LIN {X 0,Y 235.398,Z 339.465,A -85,B 0,C 180,E1 -19978.483,E2 -19978.483} C_VEL
LIN {X 0,Y 236.416,Z 340.763,A -85,B 0,C 180,E1 -19979.023,E2 -19979.023} C_VEL
LIN {X 0,Y 240.93,Z 348.91,A -85,B 0,C 180,E1 -19981.671,E2 -19981.671} C_VEL
LIN {X 0,Y 245.217,Z 358.248,A -85,B 0,C 180,E1 -19984.418,E2 -19984.418} C_VEL
LIN {X 0,Y 247.633,Z 366.708,A -85,B 0,C 180,E1 -19986.619,E2 -19986.619} C_VEL
LIN {X 0,Y 248.994,Z 374.297,A -85,B 0,C 180,E1 -19988.522,E2 -19988.522} C_VEL
LIN {X 0,Y 249.236,Z 377.337,A -85,B 0,C 180,E1 -19989.268,E2 -19989.268} C_VEL
LIN {X 0,Y 246.011,Z 387.134,A -85,B 0,C 180,E1 -19991.118,E2 -19991.118} C_VEL
LIN {X 0,Y 242.427,Z 396.773,A -85,B 0,C 180,E1 -19993.41,E2 -19993.41} C_VEL
LIN {X 0,Y 239.164,Z 404.642,A -85,B 0,C 180,E1 -19995.772,E2 -19995.772} C_VEL
LIN {X 0,Y 236.021,Z 411.635,A -85,B 0,C 180,E1 -19998.498,E2 -19998.498} C_VEL
LIN {X 0,Y 233.343,Z 416.972,A -85,B 0,C 180,E1 -20001.188,E2 -20001.188} C_VEL
LIN {X 0,Y 231.011,Z 421.302,A -85,B 0,C 180,E1 -20004.12,E2 -20004.12} C_VEL
LIN {X 0,Y 229.008,Z 424.571,A -85,B 0,C 180,E1 -20007.408,E2 -20007.408} C_VEL
LIN {X 0,Y 227.709,Z 426.199,A -85,B 0,C 180,E1 -20010.209,E2 -20010.209} C_VEL
LIN {X 0,Y 226.788,Z 426.825,A -85,B 0,C 180,E1 -20013.205,E2 -20013.205} C_VEL
LIN {X 0,Y 226.233,Z 426.352,A -85,B 0,C 180,E1 -20016.174,E2 -20016.174} C_VEL
LIN {X 0,Y 226.037,Z 424.901,A -85,B 0,C 180,E1 -20018.985,E2 -20018.985} C_VEL
LIN {X 0,Y 226.222,Z 422.441,A -85,B 0,C 180,E1 -20021.788,E2 -20021.788} C_VEL
LIN {X 0,Y 226.652,Z 419.03,A -85,B 0,C 180,E1 -20024.505,E2 -20024.505} C_VEL
LIN {X 0,Y 227.314,Z 414.656,A -85,B 0,C 180,E1 -20027.141,E2 -20027.141} C_VEL
LIN {X 0,Y 228.15,Z 409.299,A -85,B 0,C 180,E1 -20029.692,E2 -20029.692} C_VEL
LIN {X 0,Y 229.267,Z 402.802,A -85,B 0,C 180,E1 -20032.187,E2 -20032.187} C_VEL
LIN {X 0,Y 230.625,Z 395.016,A -85,B 0,C 180,E1 -20034.619,E2 -20034.619} C_VEL
LIN {X 0,Y 232.373,Z 385.49,A -85,B 0,C 180,E1 -20037.016,E2 -20037.016} C_VEL
LIN {X 0,Y 234.011,Z 375.473,A -85,B 0,C 180,E1 -20039.048,E2 -20039.048} C_VEL
LIN {X 0,Y 235.622,Z 365.003,A -85,B 0,C 180,E1 -20040.768,E2 -20040.768} C_VEL
LIN {X 0,Y 236.33,Z 359.176,A -85,B 0,C 180,E1 -20041.588,E2 -20041.588} C_VEL
LIN {X 0,Y 234.059,Z 347.494,A -85,B 0,C 180,E1 -20043.23,E2 -20043.23} C_VEL
LIN {X 0,Y 230.539,Z 335.099,A -85,B 0,C 180,E1 -20044.736,E2 -20044.736} C_VEL
LIN {X 0,Y 227.695,Z 326.123,A -85,B 0,C 180,E1 -20045.678,E2 -20045.678} C_VEL
LIN {X 0,Y 227.868,Z 326.101,A -85,B 0,C 180,E1 -20048.277,E2 -20048.277} C_VEL
LIN {X 0,Y 227.99,Z 326.086,A -85,B 0,C 180,E1 -20052.862,E2 -20052.862} C_VEL
LIN {X 0,Y 228.066,Z 326.077,A -85,B 0,C 180,E1 -20057.543,E2 -20057.543} C_VEL
LIN {X 0,Y 228.259,Z 326.056,A -85,B 0,C 180,E1 -20061.144,E2 -20061.144} C_VEL
LIN {X 0,Y 228.31,Z 326.047,A -85,B 0,C 180,E1 -20062.927,E2 -20062.927} C_VEL
LIN {X 0,Y 228.554,Z 326.015,A -85,B 0,C 180,E1 -20068.238,E2 -20068.238} C_VEL
LIN {X 0,Y 228.555,Z 326.011,A -85,B 0,C 180,E1 -20071.762,E2 -20071.762} C_VEL
LIN {X 0,Y 228.31,Z 326.043,A -85,B 0,C 180,E1 -20077.073,E2 -20077.073} C_VEL
LIN {X 0,Y 228.146,Z 326.068,A -85,B 0,C 180,E1 -20080.651,E2 -20080.651} C_VEL
LIN {X 0,Y 228.066,Z 326.076,A -85,B 0,C 180,E1 -20084.272,E2 -20084.272} C_VEL
LIN {X 0,Y 228.004,Z 326.083,A -85,B 0,C 180,E1 -20087.953,E2 -20087.953} C_VEL
LIN {X 0,Y 227.931,Z 326.092,A -85,B 0,C 180,E1 -20092.33,E2 -20092.33} C_VEL
LIN {X 0,Y 227.944,Z 326.091,A -85,B 0,C 180,E1 -20096.603,E2 -20096.603} C_VEL
LIN {X 0,Y 227.91,Z 326.094,A -85,B 0,C 180,E1 -20100.296,E2 -20100.296} C_VEL
LIN {X 0,Y 227.889,Z 326.098,A -85,B 0,C 180,E1 -20103.719,E2 -20103.719} C_VEL
LIN {X 0,Y 227.87,Z 326.099,A -85,B 0,C 180,E1 -20108.086,E2 -20108.086} C_VEL
LIN {X 0,Y 227.815,Z 326.106,A -85,B 0,C 180,E1 -20112.742,E2 -20112.742} C_VEL
LIN {X 0,Y 227.812,Z 326.104,A -85,B 0,C 180,E1 -20117.258,E2 -20117.258} C_VEL
LIN {X 0,Y 227.846,Z 326.103,A -85,B 0,C 180,E1 -20121.91,E2 -20121.91} C_VEL
LIN {X 0,Y 227.887,Z 326.095,A -85,B 0,C 180,E1 -20126.375,E2 -20126.375} C_VEL
LIN {X 0,Y 227.921,Z 326.092,A -85,B 0,C 180,E1 -20130.438,E2 -20130.438} C_VEL
LIN {X 0,Y 227.927,Z 326.09,A -85,B 0,C 180,E1 -20134.426,E2 -20134.426} C_VEL
LIN {X 0,Y 227.947,Z 326.089,A -85,B 0,C 180,E1 -20138.286,E2 -20138.286} C_VEL
LIN {X 0,Y 228.011,Z 326.081,A -85,B 0,C 180,E1 -20142.848,E2 -20142.848} C_VEL
LIN {X 0,Y 228.06,Z 326.075,A -85,B 0,C 180,E1 -20147.543,E2 -20147.543} C_VEL
LIN {X 0,Y 228.267,Z 326.052,A -85,B 0,C 180,E1 -20151.145,E2 -20151.145} C_VEL
LIN {X 0,Y 228.322,Z 326.045,A -85,B 0,C 180,E1 -20152.928,E2 -20152.928} C_VEL
LIN {X 0,Y 228.556,Z 326.011,A -85,B 0,C 180,E1 -20158.238,E2 -20158.238} C_VEL
LIN {X 0,Y 228.552,Z 326.014,A -85,B 0,C 180,E1 -20161.762,E2 -20161.762} C_VEL
LIN {X 0,Y 228.312,Z 326.044,A -85,B 0,C 180,E1 -20167.073,E2 -20167.073} C_VEL
LIN {X 0,Y 228.148,Z 326.068,A -85,B 0,C 180,E1 -20170.651,E2 -20170.651} C_VEL
LIN {X 0,Y 228.051,Z 326.075,A -85,B 0,C 180,E1 -20174.273,E2 -20174.273} C_VEL
LIN {X 0,Y 227.972,Z 326.087,A -85,B 0,C 180,E1 -20177.956,E2 -20177.956} C_VEL
LIN {X 0,Y 227.923,Z 326.091,A -85,B 0,C 180,E1 -20182.323,E2 -20182.323} C_VEL
LIN {X 0,Y 227.926,Z 326.081,A -85,B 0,C 180,E1 -20186.593,E2 -20186.593} C_VEL
LIN {X 0,Y 227.877,Z 326.097,A -85,B 0,C 180,E1 -20190.281,E2 -20190.281} C_VEL
LIN {X 0,Y 227.89,Z 326.098,A -85,B 0,C 180,E1 -20193.719,E2 -20193.719} C_VEL
LIN {X 0,Y 227.871,Z 326.102,A -85,B 0,C 180,E1 -20198.086,E2 -20198.086} C_VEL
LIN {X 0,Y 227.925,Z 326.208,A -85,B 0,C 180,E1 -20199.568,E2 -20199.568} C_VEL
LIN {X 0,Y 228.797,Z 330.781,A -85,B 0,C 180,E1 -20203.721,E2 -20203.721} C_VEL
LIN {X 0,Y 229.869,Z 336.683,A -85,B 0,C 180,E1 -20208.812,E2 -20208.812} C_VEL
LIN {X 0,Y 230.393,Z 339.72,A -85,B 0,C 180,E1 -20211.293,E2 -20211.293} C_VEL
LIN {X 0,Y 230.3,Z 342.542,A -85,B 0,C 180,E1 -20213.506,E2 -20213.506} C_VEL
LIN {X 0,Y 228.77,Z 349.178,A -85,B 0,C 180,E1 -20218.516,E2 -20218.516} C_VEL
LIN {X 0,Y 228.509,Z 350.58,A -85,B 0,C 180,E1 -20219.558,E2 -20219.558} C_VEL
LIN {X 0,Y 228.015,Z 352.382,A -85,B 0,C 180,E1 -20220.39,E2 -20220.39} C_VEL
LIN {X 0,Y 227.044,Z 355.768,A -85,B 0,C 180,E1 -20221.22,E2 -20221.22} C_VEL
LIN {X 0,Y 225.918,Z 359.881,A -85,B 0,C 180,E1 -20221.849,E2 -20221.849} C_VEL
LIN {X 0,Y 224.603,Z 365.585,A -85,B 0,C 180,E1 -20222.423,E2 -20222.423} C_VEL
LIN {X 0,Y 223.56,Z 373.659,A -85,B 0,C 180,E1 -20223.095,E2 -20223.095} C_VEL
LIN {X 0,Y 223.654,Z 377.387,A -85,B 0,C 180,E1 -20223.476,E2 -20223.476} C_VEL
LIN {X 0,Y 224.58,Z 389.329,A -85,B 0,C 180,E1 -20224.966,E2 -20224.966} C_VEL
LIN {X 0,Y 225.134,Z 401.195,A -85,B 0,C 180,E1 -20226.789,E2 -20226.789} C_VEL
LIN {X 0,Y 225.215,Z 410.46,A -85,B 0,C 180,E1 -20228.49,E2 -20228.49} C_VEL
LIN {X 0,Y 223.359,Z 420.599,A -85,B 0,C 180,E1 -20230.662,E2 -20230.662} C_VEL
LIN {X 0,Y 221.808,Z 429.212,A -85,B 0,C 180,E1 -20232.957,E2 -20232.957} C_VEL
LIN {X 0,Y 220.521,Z 437.46,A -85,B 0,C 180,E1 -20235.7,E2 -20235.7} C_VEL
LIN {X 0,Y 219.699,Z 443.077,A -85,B 0,C 180,E1 -20237.999,E2 -20237.999} C_VEL
LIN {X 0,Y 219.222,Z 448.554,A -85,B 0,C 180,E1 -20240.776,E2 -20240.776} C_VEL
LIN {X 0,Y 219.119,Z 453.231,A -85,B 0,C 180,E1 -20243.878,E2 -20243.878} C_VEL
LIN {X 0,Y 219.084,Z 455.908,A -85,B 0,C 180,E1 -20246.321,E2 -20246.321} C_VEL
LIN {X 0,Y 219.205,Z 457.414,A -85,B 0,C 180,E1 -20248.163,E2 -20248.163} C_VEL
LIN {X 0,Y 219.481,Z 458.495,A -85,B 0,C 180,E1 -20250,E2 -20250} C_VEL
LIN {X 0,Y 218.947,Z 459.218,A -85,B 0,C 180,E1 -20253.681,E2 -20253.681} C_VEL
LIN {X 0,Y 218.814,Z 458.388,A -85,B 0,C 180,E1 -20257.382,E2 -20257.382} C_VEL
LIN {X 0,Y 219.34,Z 455.952,A -85,B 0,C 180,E1 -20261.084,E2 -20261.084} C_VEL
LIN {X 0,Y 220.319,Z 453.09,A -85,B 0,C 180,E1 -20263.842,E2 -20263.842} C_VEL
LIN {X 0,Y 222.516,Z 447.791,A -85,B 0,C 180,E1 -20267.461,E2 -20267.461} C_VEL
LIN {X 0,Y 225.054,Z 441.83,A -85,B 0,C 180,E1 -20270.471,E2 -20270.471} C_VEL
LIN {X 0,Y 227.921,Z 434.999,A -85,B 0,C 180,E1 -20273.151,E2 -20273.151} C_VEL
LIN {X 0,Y 231.455,Z 426.902,A -85,B 0,C 180,E1 -20275.639,E2 -20275.639} C_VEL
LIN {X 0,Y 233.903,Z 420.63,A -85,B 0,C 180,E1 -20277.272,E2 -20277.272} C_VEL
LIN {X 0,Y 236.072,Z 410.799,A -85,B 0,C 180,E1 -20279.626,E2 -20279.626} C_VEL
LIN {X 0,Y 237.181,Z 401.09,A -85,B 0,C 180,E1 -20281.733,E2 -20281.733} C_VEL
LIN {X 0,Y 237.255,Z 388.964,A -85,B 0,C 180,E1 -20284.251,E2 -20284.251} C_VEL
LIN {X 0,Y 236.12,Z 377.783,A -85,B 0,C 180,E1 -20286.534,E2 -20286.534} C_VEL
LIN {X 0,Y 233.941,Z 366.022,A -85,B 0,C 180,E1 -20289.016,E2 -20289.016} C_VEL
LIN {X 0,Y 232.372,Z 361.024,A -85,B 0,C 180,E1 -20290.209,E2 -20290.209} C_VEL
LIN {X 0,Y 230.909,Z 357.222,A -85,B 0,C 180,E1 -20291.235,E2 -20291.235} C_VEL
LIN {X 0,Y 228.734,Z 353.288,A -85,B 0,C 180,E1 -20292.567,E2 -20292.567} C_VEL
LIN {X 0,Y 227.831,Z 351.073,A -85,B 0,C 180,E1 -20293.186,E2 -20293.186} C_VEL
LIN {X 0,Y 225.159,Z 347.328,A -85,B 0,C 180,E1 -20294.836,E2 -20294.836} C_VEL
LIN {X 0,Y 224.055,Z 344.226,A -85,B 0,C 180,E1 -20295.74,E2 -20295.74} C_VEL
LIN {X 0,Y 223.573,Z 341.782,A -85,B 0,C 180,E1 -20298.977,E2 -20298.977} C_VEL
LIN {X 0,Y 223.1,Z 338.961,A -85,B 0,C 180,E1 -20303.235,E2 -20303.235} C_VEL
LIN {X 0,Y 222.676,Z 336.61,A -85,B 0,C 180,E1 -20307.551,E2 -20307.551} C_VEL
LIN {X 0,Y 222.34,Z 334.59,A -85,B 0,C 180,E1 -20312.26,E2 -20312.26} C_VEL
LIN {X 0,Y 222.116,Z 333.25,A -85,B 0,C 180,E1 -20316.578,E2 -20316.578} C_VEL
LIN {X 0,Y 221.976,Z 332.239,A -85,B 0,C 180,E1 -20321.776,E2 -20321.776} C_VEL
LIN {X 0,Y 221.961,Z 331.908,A -85,B 0,C 180,E1 -20325.326,E2 -20325.326} C_VEL
LIN {X 0,Y 222.119,Z 331.932,A -85,B 0,C 180,E1 -20330.897,E2 -20330.897} C_VEL
LIN {X 0,Y 222.172,Z 332.099,A -85,B 0,C 180,E1 -20331.472,E2 -20331.472} C_VEL
LIN {X 0,Y 223.328,Z 334.532,A -85,B 0,C 180,E1 -20332.484,E2 -20332.484} C_VEL
LIN {X 0,Y 225.884,Z 336.883,A -85,B 0,C 180,E1 -20334.131,E2 -20334.131} C_VEL
LIN {X 0,Y 228.082,Z 340.42,A -85,B 0,C 180,E1 -20335.692,E2 -20335.692} C_VEL
LIN {X 0,Y 229.492,Z 341.637,A -85,B 0,C 180,E1 -20336.488,E2 -20336.488} C_VEL
LIN {X 0,Y 232.052,Z 345.542,A -85,B 0,C 180,E1 -20338.113,E2 -20338.113} C_VEL
LIN {X 0,Y 235.66,Z 352.189,A -85,B 0,C 180,E1 -20340.512,E2 -20340.512} C_VEL
LIN {X 0,Y 239.595,Z 360.989,A -85,B 0,C 180,E1 -20343.363,E2 -20343.363} C_VEL
LIN {X 0,Y 241.713,Z 368.228,A -85,B 0,C 180,E1 -20345.422,E2 -20345.422} C_VEL
LIN {X 0,Y 243.137,Z 376.852,A -85,B 0,C 180,E1 -20347.765,E2 -20347.765} C_VEL
LIN {X 0,Y 243.302,Z 379.462,A -85,B 0,C 180,E1 -20348.448,E2 -20348.448} C_VEL
LIN {X 0,Y 239.625,Z 389.997,A -85,B 0,C 180,E1 -20350.562,E2 -20350.562} C_VEL
LIN {X 0,Y 235.887,Z 399.194,A -85,B 0,C 180,E1 -20352.911,E2 -20352.911} C_VEL
LIN {X 0,Y 232.47,Z 406.649,A -85,B 0,C 180,E1 -20355.328,E2 -20355.328} C_VEL
LIN {X 0,Y 229.237,Z 413.358,A -85,B 0,C 180,E1 -20358.119,E2 -20358.119} C_VEL
LIN {X 0,Y 226.177,Z 418.961,A -85,B 0,C 180,E1 -20361.22,E2 -20361.22} C_VEL
LIN {X 0,Y 223.73,Z 423.003,A -85,B 0,C 180,E1 -20364.359,E2 -20364.359} C_VEL
LIN {X 0,Y 221.864,Z 425.675,A -85,B 0,C 180,E1 -20367.506,E2 -20367.506} C_VEL
LIN {X 0,Y 220.445,Z 427.13,A -85,B 0,C 180,E1 -20370.67,E2 -20370.67} C_VEL
LIN {X 0,Y 219.586,Z 427.399,A -85,B 0,C 180,E1 -20373.679,E2 -20373.679} C_VEL
LIN {X 0,Y 219.082,Z 426.619,A -85,B 0,C 180,E1 -20376.68,E2 -20376.68} C_VEL
LIN {X 0,Y 218.979,Z 424.565,A -85,B 0,C 180,E1 -20379.933,E2 -20379.933} C_VEL
LIN {X 0,Y 219.391,Z 420.77,A -85,B 0,C 180,E1 -20383.551,E2 -20383.551} C_VEL
LIN {X 0,Y 219.954,Z 416.899,A -85,B 0,C 180,E1 -20386.181,E2 -20386.181} C_VEL
LIN {X 0,Y 220.89,Z 411.056,A -85,B 0,C 180,E1 -20389.257,E2 -20389.257} C_VEL
LIN {X 0,Y 222.145,Z 403.613,A -85,B 0,C 180,E1 -20392.272,E2 -20392.272} C_VEL
LIN {X 0,Y 223.574,Z 395.754,A -85,B 0,C 180,E1 -20394.816,E2 -20394.816} C_VEL
LIN {X 0,Y 225.395,Z 386.048,A -85,B 0,C 180,E1 -20397.339,E2 -20397.339} C_VEL
LIN {X 0,Y 227.175,Z 375.569,A -85,B 0,C 180,E1 -20399.517,E2 -20399.517} C_VEL
LIN {X 0,Y 228.882,Z 364.732,A -85,B 0,C 180,E1 -20401.329,E2 -20401.329} C_VEL
LIN {X 0,Y 229.386,Z 360.768,A -85,B 0,C 180,E1 -20401.896,E2 -20401.896} C_VEL
LIN {X 0,Y 227.646,Z 350.635,A -85,B 0,C 180,E1 -20403.407,E2 -20403.407} C_VEL
LIN {X 0,Y 224.857,Z 340.173,A -85,B 0,C 180,E1 -20404.795,E2 -20404.795} C_VEL
LIN {X 0,Y 220.665,Z 326.998,A -85,B 0,C 180,E1 -20406.291,E2 -20406.291} C_VEL
LIN {X 0,Y 220.829,Z 326.979,A -85,B 0,C 180,E1 -20409.508,E2 -20409.508} C_VEL
LIN {X 0,Y 220.978,Z 326.96,A -85,B 0,C 180,E1 -20413.367,E2 -20413.367} C_VEL
LIN {X 0,Y 221.003,Z 326.959,A -85,B 0,C 180,E1 -20417.138,E2 -20417.138} C_VEL
LIN {X 0,Y 221.199,Z 326.936,A -85,B 0,C 180,E1 -20420.859,E2 -20420.859} C_VEL
LIN {X 0,Y 221.13,Z 326.939,A -85,B 0,C 180,E1 -20424.529,E2 -20424.529} C_VEL
LIN {X 0,Y 221.512,Z 326.892,A -85,B 0,C 180,E1 -20428.182,E2 -20428.182} C_VEL
LIN {X 0,Y 221.512,Z 326.888,A -85,B 0,C 180,E1 -20431.818,E2 -20431.818} C_VEL
LIN {X 0,Y 221.247,Z 326.922,A -85,B 0,C 180,E1 -20437.3,E2 -20437.3} C_VEL
LIN {X 0,Y 221.068,Z 326.947,A -85,B 0,C 180,E1 -20440.996,E2 -20440.996} C_VEL
LIN {X 0,Y 220.997,Z 326.955,A -85,B 0,C 180,E1 -20444.739,E2 -20444.739} C_VEL
LIN {X 0,Y 220.923,Z 326.966,A -85,B 0,C 180,E1 -20448.549,E2 -20448.549} C_VEL
LIN {X 0,Y 220.897,Z 326.967,A -85,B 0,C 180,E1 -20452.683,E2 -20452.683} C_VEL
LIN {X 0,Y 220.887,Z 326.969,A -85,B 0,C 180,E1 -20457.016,E2 -20457.016} C_VEL
LIN {X 0,Y 220.864,Z 326.969,A -85,B 0,C 180,E1 -20460.779,E2 -20460.779} C_VEL
LIN {X 0,Y 220.815,Z 326.977,A -85,B 0,C 180,E1 -20464.953,E2 -20464.953} C_VEL
LIN {X 0,Y 220.839,Z 326.974,A -85,B 0,C 180,E1 -20467.288,E2 -20467.288} C_VEL
LIN {X 0,Y 220.776,Z 326.986,A -85,B 0,C 180,E1 -20471.952,E2 -20471.952} C_VEL
LIN {X 0,Y 220.775,Z 326.984,A -85,B 0,C 180,E1 -20475.546,E2 -20475.546} C_VEL
LIN {X 0,Y 220.808,Z 326.979,A -85,B 0,C 180,E1 -20480.464,E2 -20480.464} C_VEL
LIN {X 0,Y 220.807,Z 326.976,A -85,B 0,C 180,E1 -20485.046,E2 -20485.046} C_VEL
LIN {X 0,Y 220.87,Z 326.974,A -85,B 0,C 180,E1 -20489.395,E2 -20489.395} C_VEL
LIN {X 0,Y 220.897,Z 326.968,A -85,B 0,C 180,E1 -20493.55,E2 -20493.55} C_VEL
LIN {X 0,Y 220.867,Z 326.973,A -85,B 0,C 180,E1 -20497.552,E2 -20497.552} C_VEL
LIN {X 0,Y 220.965,Z 326.957,A -85,B 0,C 180,E1 -20502.59,E2 -20502.59} C_VEL
LIN {X 0,Y 220.999,Z 326.957,A -85,B 0,C 180,E1 -20507.138,E2 -20507.138} C_VEL
LIN {X 0,Y 221.205,Z 326.929,A -85,B 0,C 180,E1 -20510.86,E2 -20510.86} C_VEL
LIN {X 0,Y 221.258,Z 326.924,A -85,B 0,C 180,E1 -20512.701,E2 -20512.701} C_VEL
LIN {X 0,Y 221.514,Z 326.888,A -85,B 0,C 180,E1 -20518.182,E2 -20518.182} C_VEL
LIN {X 0,Y 221.509,Z 326.891,A -85,B 0,C 180,E1 -20521.818,E2 -20521.818} C_VEL
LIN {X 0,Y 221.249,Z 326.923,A -85,B 0,C 180,E1 -20527.3,E2 -20527.3} C_VEL
LIN {X 0,Y 221.069,Z 326.947,A -85,B 0,C 180,E1 -20530.997,E2 -20530.997} C_VEL
LIN {X 0,Y 220.994,Z 326.958,A -85,B 0,C 180,E1 -20536.632,E2 -20536.632} C_VEL
LIN {X 0,Y 220.881,Z 326.97,A -85,B 0,C 180,E1 -20540.487,E2 -20540.487} C_VEL
LIN {X 0,Y 220.85,Z 326.965,A -85,B 0,C 180,E1 -20544.437,E2 -20544.437} C_VEL
LIN {X 0,Y 220.808,Z 326.973,A -85,B 0,C 180,E1 -20548.518,E2 -20548.518} C_VEL
LIN {X 0,Y 220.82,Z 326.979,A -85,B 0,C 180,E1 -20552.756,E2 -20552.756} C_VEL
LIN {X 0,Y 220.841,Z 326.975,A -85,B 0,C 180,E1 -20557.288,E2 -20557.288} C_VEL
LIN {X 0,Y 220.877,Z 327.025,A -85,B 0,C 180,E1 -20559.227,E2 -20559.227} C_VEL
LIN {X 0,Y 221.669,Z 331.227,A -85,B 0,C 180,E1 -20563.179,E2 -20563.179} C_VEL
LIN {X 0,Y 222.552,Z 336.11,A -85,B 0,C 180,E1 -20567.562,E2 -20567.562} C_VEL
LIN {X 0,Y 223.287,Z 340.125,A -85,B 0,C 180,E1 -20570.986,E2 -20570.986} C_VEL
LIN {X 0,Y 223.271,Z 342.933,A -85,B 0,C 180,E1 -20573.268,E2 -20573.268} C_VEL
LIN {X 0,Y 221.999,Z 348.253,A -85,B 0,C 180,E1 -20577.44,E2 -20577.44} C_VEL
LIN {X 0,Y 220.883,Z 353.362,A -85,B 0,C 180,E1 -20581.363,E2 -20581.363} C_VEL
LIN {X 0,Y 222.554,Z 366.713,A -85,B 0,C 180,E1 -20582.398,E2 -20582.398} C_VEL
LIN {X 0,Y 223.654,Z 377.387,A -85,B 0,C 180,E1 -20583.476,E2 -20583.476} C_VEL
LIN {X 0,Y 223.48,Z 382.834,A -85,B 0,C 180,E1 -20584.06,E2 -20584.06} C_VEL
LIN {X 0,Y 221.23,Z 391.669,A -85,B 0,C 180,E1 -20585.069,E2 -20585.069} C_VEL
LIN {X 0,Y 218.746,Z 400.184,A -85,B 0,C 180,E1 -20586.263,E2 -20586.263} C_VEL
LIN {X 0,Y 218.228,Z 405.096,A -85,B 0,C 180,E1 -20587.124,E2 -20587.124} C_VEL
LIN {X 0,Y 218.16,Z 410.813,A -85,B 0,C 180,E1 -20588.255,E2 -20588.255} C_VEL
LIN {X 0,Y 216.339,Z 420.433,A -85,B 0,C 180,E1 -20590.408,E2 -20590.408} C_VEL
LIN {X 0,Y 214.696,Z 429.244,A -85,B 0,C 180,E1 -20592.866,E2 -20592.866} C_VEL
LIN {X 0,Y 213.42,Z 437.397,A -85,B 0,C 180,E1 -20595.701,E2 -20595.701} C_VEL
LIN {X 0,Y 212.514,Z 443.938,A -85,B 0,C 180,E1 -20598.555,E2 -20598.555} C_VEL
LIN {X 0,Y 212.084,Z 449.114,A -85,B 0,C 180,E1 -20601.424,E2 -20601.424} C_VEL
LIN {X 0,Y 212.069,Z 453.087,A -85,B 0,C 180,E1 -20604.294,E2 -20604.294} C_VEL
LIN {X 0,Y 212.021,Z 455.078,A -85,B 0,C 180,E1 -20606.199,E2 -20606.199} C_VEL
LIN {X 0,Y 212.127,Z 456.63,A -85,B 0,C 180,E1 -20608.101,E2 -20608.101} C_VEL
LIN {X 0,Y 212.423,Z 457.773,A -85,B 0,C 180,E1 -20610,E2 -20610} C_VEL
LIN {X 0,Y 212.012,Z 458.413,A -85,B 0,C 180,E1 -20611.9,E2 -20611.9} C_VEL
LIN {X 0,Y 211.738,Z 458.548,A -85,B 0,C 180,E1 -20615.275,E2 -20615.275} C_VEL
LIN {X 0,Y 211.732,Z 457.909,A -85,B 0,C 180,E1 -20617.63,E2 -20617.63} C_VEL
LIN {X 0,Y 211.925,Z 456.976,A -85,B 0,C 180,E1 -20619.545,E2 -20619.545} C_VEL
LIN {X 0,Y 212.937,Z 453.896,A -85,B 0,C 180,E1 -20623.358,E2 -20623.358} C_VEL
LIN {X 0,Y 215.066,Z 449.218,A -85,B 0,C 180,E1 -20627.104,E2 -20627.104} C_VEL
LIN {X 0,Y 217.335,Z 444.513,A -85,B 0,C 180,E1 -20629.849,E2 -20629.849} C_VEL
LIN {X 0,Y 220.345,Z 437.609,A -85,B 0,C 180,E1 -20633,E2 -20633} C_VEL
LIN {X 0,Y 223.809,Z 430.287,A -85,B 0,C 180,E1 -20635.58,E2 -20635.58} C_VEL
LIN {X 0,Y 227.64,Z 421.393,A -85,B 0,C 180,E1 -20638.088,E2 -20638.088} C_VEL
LIN {X 0,Y 229.652,Z 413.383,A -85,B 0,C 180,E1 -20640.132,E2 -20640.132} C_VEL
LIN {X 0,Y 231.265,Z 402.662,A -85,B 0,C 180,E1 -20642.643,E2 -20642.643} C_VEL
LIN {X 0,Y 231.615,Z 391.014,A -85,B 0,C 180,E1 -20645.207,E2 -20645.207} C_VEL
LIN {X 0,Y 230.806,Z 379.91,A -85,B 0,C 180,E1 -20647.655,E2 -20647.655} C_VEL
LIN {X 0,Y 229.007,Z 369.105,A -85,B 0,C 180,E1 -20650.126,E2 -20650.126} C_VEL
LIN {X 0,Y 227.528,Z 364.032,A -85,B 0,C 180,E1 -20651.491,E2 -20651.491} C_VEL
LIN {X 0,Y 224.536,Z 357.075,A -85,B 0,C 180,E1 -20653.75,E2 -20653.75} C_VEL
LIN {X 0,Y 221.85,Z 352.697,A -85,B 0,C 180,E1 -20655.661,E2 -20655.661} C_VEL
LIN {X 0,Y 220.851,Z 350.102,A -85,B 0,C 180,E1 -20656.527,E2 -20656.527} C_VEL
LIN {X 0,Y 218.008,Z 346.348,A -85,B 0,C 180,E1 -20658.741,E2 -20658.741} C_VEL
LIN {X 0,Y 216.557,Z 342.773,A -85,B 0,C 180,E1 -20660.206,E2 -20660.206} C_VEL
LIN {X 0,Y 216.116,Z 340.043,A -85,B 0,C 180,E1 -20664.39,E2 -20664.39} C_VEL
LIN {X 0,Y 215.732,Z 337.931,A -85,B 0,C 180,E1 -20668.584,E2 -20668.584} C_VEL
LIN {X 0,Y 215.461,Z 336.232,A -85,B 0,C 180,E1 -20672.828,E2 -20672.828} C_VEL
LIN {X 0,Y 215.237,Z 335.02,A -85,B 0,C 180,E1 -20676.931,E2 -20676.931} C_VEL
LIN {X 0,Y 215.114,Z 334.152,A -85,B 0,C 180,E1 -20681.347,E2 -20681.347} C_VEL
LIN {X 0,Y 215.08,Z 333.724,A -85,B 0,C 180,E1 -20685.814,E2 -20685.814} C_VEL
LIN {X 0,Y 215.118,Z 333.803,A -85,B 0,C 180,E1 -20686.834,E2 -20686.834} C_VEL
LIN {X 0,Y 216.296,Z 336.121,A -85,B 0,C 180,E1 -20688.235,E2 -20688.235} C_VEL
LIN {X 0,Y 219.069,Z 338.321,A -85,B 0,C 180,E1 -20690.596,E2 -20690.596} C_VEL
LIN {X 0,Y 219.629,Z 338.806,A -85,B 0,C 180,E1 -20691.025,E2 -20691.025} C_VEL
LIN {X 0,Y 221.193,Z 341.55,A -85,B 0,C 180,E1 -20692.468,E2 -20692.468} C_VEL
LIN {X 0,Y 222.877,Z 343.176,A -85,B 0,C 180,E1 -20693.663,E2 -20693.663} C_VEL
LIN {X 0,Y 223.988,Z 345.26,A -85,B 0,C 180,E1 -20694.599,E2 -20694.599} C_VEL
LIN {X 0,Y 226.608,Z 348.645,A -85,B 0,C 180,E1 -20696.444,E2 -20696.444} C_VEL
LIN {X 0,Y 229.122,Z 352.769,A -85,B 0,C 180,E1 -20698.242,E2 -20698.242} C_VEL
LIN {X 0,Y 232.587,Z 360.357,A -85,B 0,C 180,E1 -20701.038,E2 -20701.038} C_VEL
LIN {X 0,Y 235.227,Z 367.443,A -85,B 0,C 180,E1 -20703.426,E2 -20703.426} C_VEL
LIN {X 0,Y 236.756,Z 374.549,A -85,B 0,C 180,E1 -20705.536,E2 -20705.536} C_VEL
LIN {X 0,Y 237.386,Z 380.371,A -85,B 0,C 180,E1 -20707.228,E2 -20707.228} C_VEL
LIN {X 0,Y 237.398,Z 381.908,A -85,B 0,C 180,E1 -20707.655,E2 -20707.655} C_VEL
LIN {X 0,Y 233.856,Z 391.243,A -85,B 0,C 180,E1 -20709.607,E2 -20709.607} C_VEL
LIN {X 0,Y 229.922,Z 400.314,A -85,B 0,C 180,E1 -20712,E2 -20712} C_VEL
LIN {X 0,Y 226.478,Z 407.432,A -85,B 0,C 180,E1 -20714.374,E2 -20714.374} C_VEL
LIN {X 0,Y 222.926,Z 414.218,A -85,B 0,C 180,E1 -20717.288,E2 -20717.288} C_VEL
LIN {X 0,Y 219.543,Z 419.931,A -85,B 0,C 180,E1 -20720.618,E2 -20720.618} C_VEL
LIN {X 0,Y 217.738,Z 422.765,A -85,B 0,C 180,E1 -20722.788,E2 -20722.788} C_VEL
LIN {X 0,Y 216.192,Z 424.925,A -85,B 0,C 180,E1 -20724.999,E2 -20724.999} C_VEL
LIN {X 0,Y 214.571,Z 426.835,A -85,B 0,C 180,E1 -20727.827,E2 -20727.827} C_VEL
LIN {X 0,Y 213.228,Z 427.884,A -85,B 0,C 180,E1 -20731.022,E2 -20731.022} C_VEL
LIN {X 0,Y 212.383,Z 427.814,A -85,B 0,C 180,E1 -20734.232,E2 -20734.232} C_VEL
LIN {X 0,Y 211.969,Z 426.715,A -85,B 0,C 180,E1 -20737.274,E2 -20737.274} C_VEL
LIN {X 0,Y 211.912,Z 424.62,A -85,B 0,C 180,E1 -20740.289,E2 -20740.289} C_VEL
LIN {X 0,Y 212.387,Z 420.563,A -85,B 0,C 180,E1 -20744.019,E2 -20744.019} C_VEL
LIN {X 0,Y 213.094,Z 415.77,A -85,B 0,C 180,E1 -20747.137,E2 -20747.137} C_VEL
LIN {X 0,Y 214.158,Z 409.36,A -85,B 0,C 180,E1 -20750.335,E2 -20750.335} C_VEL
LIN {X 0,Y 215.376,Z 402.737,A -85,B 0,C 180,E1 -20752.956,E2 -20752.956} C_VEL
LIN {X 0,Y 216.997,Z 393.925,A -85,B 0,C 180,E1 -20755.755,E2 -20755.755} C_VEL
LIN {X 0,Y 218.922,Z 383.945,A -85,B 0,C 180,E1 -20758.285,E2 -20758.285} C_VEL
LIN {X 0,Y 220.749,Z 373.38,A -85,B 0,C 180,E1 -20760.43,E2 -20760.43} C_VEL
LIN {X 0,Y 222.439,Z 362.413,A -85,B 0,C 180,E1 -20762.21,E2 -20762.21} C_VEL
LIN {X 0,Y 221.944,Z 357.936,A -85,B 0,C 180,E1 -20762.922,E2 -20762.922} C_VEL
LIN {X 0,Y 219.782,Z 347.789,A -85,B 0,C 180,E1 -20764.425,E2 -20764.425} C_VEL
LIN {X 0,Y 216.14,Z 335.531,A -85,B 0,C 180,E1 -20766.019,E2 -20766.019} C_VEL
LIN {X 0,Y 213.656,Z 327.873,A -85,B 0,C 180,E1 -20766.883,E2 -20766.883} C_VEL
LIN {X 0,Y 213.787,Z 327.856,A -85,B 0,C 180,E1 -20770.808,E2 -20770.808} C_VEL
LIN {X 0,Y 213.904,Z 327.841,A -85,B 0,C 180,E1 -20774.761,E2 -20774.761} C_VEL
LIN {X 0,Y 214.122,Z 327.814,A -85,B 0,C 180,E1 -20779.955,E2 -20779.955} C_VEL
LIN {X 0,Y 214.188,Z 327.807,A -85,B 0,C 180,E1 -20782.458,E2 -20782.458} C_VEL
LIN {X 0,Y 214.445,Z 327.772,A -85,B 0,C 180,E1 -20788.122,E2 -20788.122} C_VEL
LIN {X 0,Y 214.551,Z 327.755,A -85,B 0,C 180,E1 -20790,E2 -20790} C_VEL
LIN {X 0,Y 214.445,Z 327.768,A -85,B 0,C 180,E1 -20791.878,E2 -20791.878} C_VEL
LIN {X 0,Y 214.188,Z 327.801,A -85,B 0,C 180,E1 -20797.542,E2 -20797.542} C_VEL
LIN {X 0,Y 214,Z 327.827,A -85,B 0,C 180,E1 -20801.364,E2 -20801.364} C_VEL
LIN {X 0,Y 213.935,Z 327.833,A -85,B 0,C 180,E1 -20805.237,E2 -20805.237} C_VEL
LIN {X 0,Y 213.841,Z 327.846,A -85,B 0,C 180,E1 -20809.187,E2 -20809.187} C_VEL
LIN {X 0,Y 213.848,Z 327.843,A -85,B 0,C 180,E1 -20813.227,E2 -20813.227} C_VEL
LIN {X 0,Y 213.83,Z 327.848,A -85,B 0,C 180,E1 -20817.45,E2 -20817.45} C_VEL
LIN {X 0,Y 213.78,Z 327.853,A -85,B 0,C 180,E1 -20821.736,E2 -20821.736} C_VEL
LIN {X 0,Y 213.753,Z 327.858,A -85,B 0,C 180,E1 -20826.287,E2 -20826.287} C_VEL
LIN {X 0,Y 213.717,Z 327.861,A -85,B 0,C 180,E1 -20831.124,E2 -20831.124} C_VEL
LIN {X 0,Y 213.709,Z 327.865,A -85,B 0,C 180,E1 -20833.678,E2 -20833.678} C_VEL
LIN {X 0,Y 213.707,Z 327.86,A -85,B 0,C 180,E1 -20836.344,E2 -20836.344} C_VEL
LIN {X 0,Y 213.718,Z 327.861,A -85,B 0,C 180,E1 -20839.143,E2 -20839.143} C_VEL
LIN {X 0,Y 213.747,Z 327.858,A -85,B 0,C 180,E1 -20843.712,E2 -20843.712} C_VEL
LIN {X 0,Y 213.797,Z 327.852,A -85,B 0,C 180,E1 -20848.725,E2 -20848.725} C_VEL
LIN {X 0,Y 213.828,Z 327.845,A -85,B 0,C 180,E1 -20852.604,E2 -20852.604} C_VEL
LIN {X 0,Y 213.821,Z 327.85,A -85,B 0,C 180,E1 -20856.974,E2 -20856.974} C_VEL
LIN {X 0,Y 213.924,Z 327.835,A -85,B 0,C 180,E1 -20862.802,E2 -20862.802} C_VEL
LIN {X 0,Y 213.94,Z 327.835,A -85,B 0,C 180,E1 -20866.706,E2 -20866.706} C_VEL
LIN {X 0,Y 214.143,Z 327.807,A -85,B 0,C 180,E1 -20870.555,E2 -20870.555} C_VEL
LIN {X 0,Y 214.099,Z 327.815,A -85,B 0,C 180,E1 -20874.349,E2 -20874.349} C_VEL
LIN {X 0,Y 214.447,Z 327.768,A -85,B 0,C 180,E1 -20878.122,E2 -20878.122} C_VEL
LIN {X 0,Y 214.549,Z 327.757,A -85,B 0,C 180,E1 -20880,E2 -20880} C_VEL
LIN {X 0,Y 214.442,Z 327.771,A -85,B 0,C 180,E1 -20881.878,E2 -20881.878} C_VEL
LIN {X 0,Y 214.19,Z 327.802,A -85,B 0,C 180,E1 -20887.542,E2 -20887.542} C_VEL
LIN {X 0,Y 214,Z 327.826,A -85,B 0,C 180,E1 -20891.365,E2 -20891.365} C_VEL
LIN {X 0,Y 213.915,Z 327.836,A -85,B 0,C 180,E1 -20895.239,E2 -20895.239} C_VEL
LIN {X 0,Y 213.823,Z 327.848,A -85,B 0,C 180,E1 -20899.189,E2 -20899.189} C_VEL
LIN {X 0,Y 213.805,Z 327.844,A -85,B 0,C 180,E1 -20903.232,E2 -20903.232} C_VEL
LIN {X 0,Y 213.79,Z 327.84,A -85,B 0,C 180,E1 -20907.428,E2 -20907.428} C_VEL
LIN {X 0,Y 213.763,Z 327.856,A -85,B 0,C 180,E1 -20911.739,E2 -20911.739} C_VEL
LIN {X 0,Y 213.754,Z 327.859,A -85,B 0,C 180,E1 -20916.287,E2 -20916.287} C_VEL
LIN {X 0,Y 213.87,Z 327.913,A -85,B 0,C 180,E1 -20918.938,E2 -20918.938} C_VEL
LIN {X 0,Y 214.785,Z 333.077,A -85,B 0,C 180,E1 -20923.956,E2 -20923.956} C_VEL
LIN {X 0,Y 215.72,Z 338.11,A -85,B 0,C 180,E1 -20928.532,E2 -20928.532} C_VEL
LIN {X 0,Y 216.275,Z 341.952,A -85,B 0,C 180,E1 -20931.872,E2 -20931.872} C_VEL
LIN {X 0,Y 215.942,Z 344.682,A -85,B 0,C 180,E1 -20934.138,E2 -20934.138} C_VEL
LIN {X 0,Y 214.312,Z 351.273,A -85,B 0,C 180,E1 -20939.449,E2 -20939.449} C_VEL
LIN {X 0,Y 213.947,Z 353.094,A -85,B 0,C 180,E1 -20940.732,E2 -20940.732} C_VEL
LIN {X 0,Y 215.692,Z 367.02,A -85,B 0,C 180,E1 -20941.859,E2 -20941.859} C_VEL
LIN {X 0,Y 216.982,Z 380.237,A -85,B 0,C 180,E1 -20943.298,E2 -20943.298} C_VEL
LIN {X 0,Y 217.823,Z 392.969,A -85,B 0,C 180,E1 -20945.045,E2 -20945.045} C_VEL
LIN {X 0,Y 218.228,Z 405.096,A -85,B 0,C 180,E1 -20947.124,E2 -20947.124} C_VEL
LIN {X 0,Y 217.875,Z 408.295,A -85,B 0,C 180,E1 -20947.723,E2 -20947.723} C_VEL
LIN {X 0,Y 216.128,Z 412.858,A -85,B 0,C 180,E1 -20948.602,E2 -20948.602} C_VEL
LIN {X 0,Y 210.032,Z 422.579,A -85,B 0,C 180,E1 -20950.788,E2 -20950.788} C_VEL
LIN {X 0,Y 208.157,Z 426.539,A -85,B 0,C 180,E1 -20951.916,E2 -20951.916} C_VEL
LIN {X 0,Y 207.829,Z 427.837,A -85,B 0,C 180,E1 -20952.327,E2 -20952.327} C_VEL
LIN {X 0,Y 206.517,Z 436.028,A -85,B 0,C 180,E1 -20955.212,E2 -20955.212} C_VEL
LIN {X 0,Y 205.509,Z 442.701,A -85,B 0,C 180,E1 -20958.159,E2 -20958.159} C_VEL
LIN {X 0,Y 205.057,Z 448.019,A -85,B 0,C 180,E1 -20961.128,E2 -20961.128} C_VEL
LIN {X 0,Y 205.003,Z 452.733,A -85,B 0,C 180,E1 -20964.616,E2 -20964.616} C_VEL
LIN {X 0,Y 205.049,Z 455.836,A -85,B 0,C 180,E1 -20968.036,E2 -20968.036} C_VEL
LIN {X 0,Y 205.364,Z 457.035,A -85,B 0,C 180,E1 -20970,E2 -20970} C_VEL
LIN {X 0,Y 204.801,Z 458.057,A -85,B 0,C 180,E1 -20973.936,E2 -20973.936} C_VEL
LIN {X 0,Y 204.659,Z 457.435,A -85,B 0,C 180,E1 -20977.895,E2 -20977.895} C_VEL
LIN {X 0,Y 205.341,Z 455.32,A -85,B 0,C 180,E1 -20981.85,E2 -20981.85} C_VEL
LIN {X 0,Y 206.487,Z 452.679,A -85,B 0,C 180,E1 -20984.79,E2 -20984.79} C_VEL
LIN {X 0,Y 208.247,Z 449.112,A -85,B 0,C 180,E1 -20987.682,E2 -20987.682} C_VEL
LIN {X 0,Y 210.625,Z 444.626,A -85,B 0,C 180,E1 -20990.479,E2 -20990.479} C_VEL
LIN {X 0,Y 213.297,Z 438.957,A -85,B 0,C 180,E1 -20993.291,E2 -20993.291} C_VEL
LIN {X 0,Y 216.813,Z 432.075,A -85,B 0,C 180,E1 -20995.951,E2 -20995.951} C_VEL
LIN {X 0,Y 220.817,Z 423.709,A -85,B 0,C 180,E1 -20998.517,E2 -20998.517} C_VEL
LIN {X 0,Y 223.23,Z 415.934,A -85,B 0,C 180,E1 -21000.664,E2 -21000.664} C_VEL
LIN {X 0,Y 225.129,Z 406.202,A -85,B 0,C 180,E1 -21003.113,E2 -21003.113} C_VEL
LIN {X 0,Y 225.965,Z 395.597,A -85,B 0,C 180,E1 -21005.635,E2 -21005.635} C_VEL
LIN {X 0,Y 225.809,Z 385.855,A -85,B 0,C 180,E1 -21007.934,E2 -21007.934} C_VEL
LIN {X 0,Y 224.626,Z 374.332,A -85,B 0,C 180,E1 -21010.707,E2 -21010.707} C_VEL
LIN {X 0,Y 223.243,Z 368.761,A -85,B 0,C 180,E1 -21012.284,E2 -21012.284} C_VEL
LIN {X 0,Y 220.878,Z 362.624,A -85,B 0,C 180,E1 -21014.428,E2 -21014.428} C_VEL
LIN {X 0,Y 218.566,Z 358.596,A -85,B 0,C 180,E1 -21016.264,E2 -21016.264} C_VEL
LIN {X 0,Y 217.601,Z 355.911,A -85,B 0,C 180,E1 -21017.293,E2 -21017.293} C_VEL
LIN {X 0,Y 215.1,Z 352.144,A -85,B 0,C 180,E1 -21019.505,E2 -21019.505} C_VEL
LIN {X 0,Y 213.754,Z 348.65,A -85,B 0,C 180,E1 -21021.16,E2 -21021.16} C_VEL
LIN {X 0,Y 209.961,Z 343.025,A -85,B 0,C 180,E1 -21026.043,E2 -21026.043} C_VEL
LIN {X 0,Y 208.83,Z 339.642,A -85,B 0,C 180,E1 -21028.839,E2 -21028.839} C_VEL
LIN {X 0,Y 208.633,Z 338.425,A -85,B 0,C 180,E1 -21031.861,E2 -21031.861} C_VEL
LIN {X 0,Y 208.417,Z 337.085,A -85,B 0,C 180,E1 -21036.13,E2 -21036.13} C_VEL
LIN {X 0,Y 208.334,Z 336.704,A -85,B 0,C 180,E1 -21038.478,E2 -21038.478} C_VEL
LIN {X 0,Y 211.099,Z 339.682,A -85,B 0,C 180,E1 -21044.306,E2 -21044.306} C_VEL
LIN {X 0,Y 212.956,Z 340.706,A -85,B 0,C 180,E1 -21046.509,E2 -21046.509} C_VEL
LIN {X 0,Y 214.269,Z 343.078,A -85,B 0,C 180,E1 -21048.222,E2 -21048.222} C_VEL
LIN {X 0,Y 216.922,Z 345.438,A -85,B 0,C 180,E1 -21050.677,E2 -21050.677} C_VEL
LIN {X 0,Y 218.913,Z 348.615,A -85,B 0,C 180,E1 -21052.622,E2 -21052.622} C_VEL
LIN {X 0,Y 219.475,Z 349.173,A -85,B 0,C 180,E1 -21053.066,E2 -21053.066} C_VEL
LIN {X 0,Y 224.512,Z 357.065,A -85,B 0,C 180,E1 -21057.275,E2 -21057.275} C_VEL
LIN {X 0,Y 227.426,Z 363.885,A -85,B 0,C 180,E1 -21060,E2 -21060} C_VEL
LIN {X 0,Y 229.945,Z 371.09,A -85,B 0,C 180,E1 -21062.627,E2 -21062.627} C_VEL
LIN {X 0,Y 231.169,Z 377.993,A -85,B 0,C 180,E1 -21064.87,E2 -21064.87} C_VEL
LIN {X 0,Y 231.617,Z 383.394,A -85,B 0,C 180,E1 -21066.533,E2 -21066.533} C_VEL
LIN {X 0,Y 230.742,Z 386.378,A -85,B 0,C 180,E1 -21067.218,E2 -21067.218} C_VEL
LIN {X 0,Y 226.848,Z 395.58,A -85,B 0,C 180,E1 -21069.36,E2 -21069.36} C_VEL
LIN {X 0,Y 222.671,Z 404.187,A -85,B 0,C 180,E1 -21071.919,E2 -21071.919} C_VEL
LIN {X 0,Y 218.464,Z 411.978,A -85,B 0,C 180,E1 -21074.913,E2 -21074.913} C_VEL
LIN {X 0,Y 215.279,Z 417.377,A -85,B 0,C 180,E1 -21077.644,E2 -21077.644} C_VEL
LIN {X 0,Y 212.66,Z 421.405,A -85,B 0,C 180,E1 -21080.304,E2 -21080.304} C_VEL
LIN {X 0,Y 209.951,Z 425.088,A -85,B 0,C 180,E1 -21083.684,E2 -21083.684} C_VEL
LIN {X 0,Y 208.471,Z 426.801,A -85,B 0,C 180,E1 -21085.993,E2 -21085.993} C_VEL
LIN {X 0,Y 207.218,Z 427.957,A -85,B 0,C 180,E1 -21088.348,E2 -21088.348} C_VEL
LIN {X 0,Y 205.993,Z 428.579,A -85,B 0,C 180,E1 -21091.466,E2 -21091.466} C_VEL
LIN {X 0,Y 205.192,Z 428.169,A -85,B 0,C 180,E1 -21094.712,E2 -21094.712} C_VEL
LIN {X 0,Y 204.818,Z 426.573,A -85,B 0,C 180,E1 -21098.144,E2 -21098.144} C_VEL
LIN {X 0,Y 204.988,Z 423.297,A -85,B 0,C 180,E1 -21102.046,E2 -21102.046} C_VEL
LIN {X 0,Y 205.452,Z 419.816,A -85,B 0,C 180,E1 -21104.875,E2 -21104.875} C_VEL
LIN {X 0,Y 206.134,Z 415.385,A -85,B 0,C 180,E1 -21107.668,E2 -21107.668} C_VEL
LIN {X 0,Y 207.074,Z 409.903,A -85,B 0,C 180,E1 -21110.431,E2 -21110.431} C_VEL
LIN {X 0,Y 208.335,Z 403.25,A -85,B 0,C 180,E1 -21113.15,E2 -21113.15} C_VEL
LIN {X 0,Y 209.97,Z 394.591,A -85,B 0,C 180,E1 -21115.992,E2 -21115.992} C_VEL
LIN {X 0,Y 211.958,Z 384.46,A -85,B 0,C 180,E1 -21118.646,E2 -21118.646} C_VEL
LIN {X 0,Y 213.817,Z 374.023,A -85,B 0,C 180,E1 -21120.833,E2 -21120.833} C_VEL
LIN {X 0,Y 215.552,Z 363.178,A -85,B 0,C 180,E1 -21122.651,E2 -21122.651} C_VEL
LIN {X 0,Y 214.352,Z 355.024,A -85,B 0,C 180,E1 -21123.99,E2 -21123.99} C_VEL
LIN {X 0,Y 211.768,Z 345.003,A -85,B 0,C 180,E1 -21125.492,E2 -21125.492} C_VEL
LIN {X 0,Y 207.629,Z 332.028,A -85,B 0,C 180,E1 -21127.169,E2 -21127.169} C_VEL
LIN {X 0,Y 206.624,Z 328.749,A -85,B 0,C 180,E1 -21127.541,E2 -21127.541} C_VEL
LIN {X 0,Y 206.822,Z 328.722,A -85,B 0,C 180,E1 -21132.192,E2 -21132.192} C_VEL
LIN {X 0,Y 206.881,Z 328.715,A -85,B 0,C 180,E1 -21136.243,E2 -21136.243} C_VEL
LIN {X 0,Y 207.08,Z 328.692,A -85,B 0,C 180,E1 -21140.23,E2 -21140.23} C_VEL
LIN {X 0,Y 207.053,Z 328.691,A -85,B 0,C 180,E1 -21144.155,E2 -21144.155} C_VEL
LIN {X 0,Y 207.381,Z 328.652,A -85,B 0,C 180,E1 -21148.058,E2 -21148.058} C_VEL
LIN {X 0,Y 207.516,Z 328.632,A -85,B 0,C 180,E1 -21150,E2 -21150} C_VEL
LIN {X 0,Y 207.381,Z 328.648,A -85,B 0,C 180,E1 -21151.942,E2 -21151.942} C_VEL
LIN {X 0,Y 207.132,Z 328.68,A -85,B 0,C 180,E1 -21157.8,E2 -21157.8} C_VEL
LIN {X 0,Y 206.926,Z 328.708,A -85,B 0,C 180,E1 -21161.758,E2 -21161.758} C_VEL
LIN {X 0,Y 206.868,Z 328.714,A -85,B 0,C 180,E1 -21165.771,E2 -21165.771} C_VEL
LIN {X 0,Y 206.785,Z 328.726,A -85,B 0,C 180,E1 -21169.869,E2 -21169.869} C_VEL
LIN {X 0,Y 206.764,Z 328.728,A -85,B 0,C 180,E1 -21174.072,E2 -21174.072} C_VEL
LIN {X 0,Y 206.745,Z 328.731,A -85,B 0,C 180,E1 -21178.419,E2 -21178.419} C_VEL
LIN {X 0,Y 206.71,Z 328.734,A -85,B 0,C 180,E1 -21182.956,E2 -21182.956} C_VEL
LIN {X 0,Y 206.723,Z 328.733,A -85,B 0,C 180,E1 -21185.321,E2 -21185.321} C_VEL
LIN {X 0,Y 206.667,Z 328.741,A -85,B 0,C 180,E1 -21190.25,E2 -21190.25} C_VEL
LIN {X 0,Y 206.635,Z 328.745,A -85,B 0,C 180,E1 -21195.582,E2 -21195.582} C_VEL
LIN {X 0,Y 206.662,Z 328.743,A -85,B 0,C 180,E1 -21199.749,E2 -21199.749} C_VEL
LIN {X 0,Y 206.717,Z 328.73,A -85,B 0,C 180,E1 -21204.692,E2 -21204.692} C_VEL
LIN {X 0,Y 206.726,Z 328.735,A -85,B 0,C 180,E1 -21209.34,E2 -21209.34} C_VEL
LIN {X 0,Y 206.733,Z 328.732,A -85,B 0,C 180,E1 -21213.772,E2 -21213.772} C_VEL
LIN {X 0,Y 206.738,Z 328.731,A -85,B 0,C 180,E1 -21218.041,E2 -21218.041} C_VEL
LIN {X 0,Y 206.87,Z 328.712,A -85,B 0,C 180,E1 -21222.196,E2 -21222.196} C_VEL
LIN {X 0,Y 206.882,Z 328.713,A -85,B 0,C 180,E1 -21226.244,E2 -21226.244} C_VEL
LIN {X 0,Y 207.102,Z 328.683,A -85,B 0,C 180,E1 -21230.231,E2 -21230.231} C_VEL
LIN {X 0,Y 207.061,Z 328.691,A -85,B 0,C 180,E1 -21234.156,E2 -21234.156} C_VEL
LIN {X 0,Y 207.383,Z 328.648,A -85,B 0,C 180,E1 -21238.058,E2 -21238.058} C_VEL
LIN {X 0,Y 207.514,Z 328.634,A -85,B 0,C 180,E1 -21240,E2 -21240} C_VEL
LIN {X 0,Y 207.378,Z 328.651,A -85,B 0,C 180,E1 -21241.942,E2 -21241.942} C_VEL
LIN {X 0,Y 207.134,Z 328.681,A -85,B 0,C 180,E1 -21247.8,E2 -21247.8} C_VEL
LIN {X 0,Y 206.924,Z 328.707,A -85,B 0,C 180,E1 -21251.759,E2 -21251.759} C_VEL
LIN {X 0,Y 206.848,Z 328.716,A -85,B 0,C 180,E1 -21255.772,E2 -21255.772} C_VEL
LIN {X 0,Y 206.859,Z 328.717,A -85,B 0,C 180,E1 -21257.955,E2 -21257.955} C_VEL
LIN {X 0,Y 206.748,Z 328.723,A -85,B 0,C 180,E1 -21263.391,E2 -21263.391} C_VEL
LIN {X 0,Y 206.691,Z 328.728,A -85,B 0,C 180,E1 -21268.427,E2 -21268.427} C_VEL
LIN {X 0,Y 206.704,Z 328.737,A -85,B 0,C 180,E1 -21272.957,E2 -21272.957} C_VEL
LIN {X 0,Y 206.74,Z 328.734,A -85,B 0,C 180,E1 -21277.727,E2 -21277.727} C_VEL
LIN {X 0,Y 206.844,Z 328.96,A -85,B 0,C 180,E1 -21278.849,E2 -21278.849} C_VEL
LIN {X 0,Y 207.725,Z 333.796,A -85,B 0,C 180,E1 -21283.686,E2 -21283.686} C_VEL
LIN {X 0,Y 208.793,Z 339.544,A -85,B 0,C 180,E1 -21289.092,E2 -21289.092} C_VEL
LIN {X 0,Y 209.23,Z 342.48,A -85,B 0,C 180,E1 -21291.732,E2 -21291.732} C_VEL
LIN {X 0,Y 208.91,Z 344.934,A -85,B 0,C 180,E1 -21293.843,E2 -21293.843} C_VEL
LIN {X 0,Y 207.706,Z 349.636,A -85,B 0,C 180,E1 -21297.77,E2 -21297.77} C_VEL
LIN {X 0,Y 207.028,Z 352.354,A -85,B 0,C 180,E1 -21300.023,E2 -21300.023} C_VEL
LIN {X 0,Y 208.629,Z 365.683,A -85,B 0,C 180,E1 -21301.146,E2 -21301.146} C_VEL
LIN {X 0,Y 209.918,Z 379.126,A -85,B 0,C 180,E1 -21302.644,E2 -21302.644} C_VEL
LIN {X 0,Y 210.723,Z 391.003,A -85,B 0,C 180,E1 -21304.305,E2 -21304.305} C_VEL
LIN {X 0,Y 211.127,Z 402.135,A -85,B 0,C 180,E1 -21306.195,E2 -21306.195} C_VEL
LIN {X 0,Y 211.102,Z 411.075,A -85,B 0,C 180,E1 -21308.004,E2 -21308.004} C_VEL
LIN {X 0,Y 209.13,Z 421.011,A -85,B 0,C 180,E1 -21310.363,E2 -21310.363} C_VEL
LIN {X 0,Y 207.829,Z 427.837,A -85,B 0,C 180,E1 -21312.327,E2 -21312.327} C_VEL
LIN {X 0,Y 206.521,Z 431.585,A -85,B 0,C 180,E1 -21313.558,E2 -21313.558} C_VEL
LIN {X 0,Y 201.158,Z 438.976,A -85,B 0,C 180,E1 -21316.5,E2 -21316.5} C_VEL
LIN {X 0,Y 198.708,Z 442.732,A -85,B 0,C 180,E1 -21318.373,E2 -21318.373} C_VEL
LIN {X 0,Y 198.201,Z 444.533,A -85,B 0,C 180,E1 -21319.375,E2 -21319.375} C_VEL
LIN {X 0,Y 197.885,Z 449.879,A -85,B 0,C 180,E1 -21322.859,E2 -21322.859} C_VEL
LIN {X 0,Y 197.961,Z 451.952,A -85,B 0,C 180,E1 -21324.563,E2 -21324.563} C_VEL
LIN {X 0,Y 197.972,Z 455.041,A -85,B 0,C 180,E1 -21327.966,E2 -21327.966} C_VEL
LIN {X 0,Y 198.305,Z 456.294,A -85,B 0,C 180,E1 -21330,E2 -21330} C_VEL
LIN {X 0,Y 197.729,Z 457.429,A -85,B 0,C 180,E1 -21334.077,E2 -21334.077} C_VEL
LIN {X 0,Y 197.57,Z 457.404,A -85,B 0,C 180,E1 -21336.126,E2 -21336.126} C_VEL
LIN {X 0,Y 197.864,Z 456.155,A -85,B 0,C 180,E1 -21340.23,E2 -21340.23} C_VEL
LIN {X 0,Y 199.069,Z 453.41,A -85,B 0,C 180,E1 -21344.308,E2 -21344.308} C_VEL
LIN {X 0,Y 200.821,Z 450.305,A -85,B 0,C 180,E1 -21347.306,E2 -21347.306} C_VEL
LIN {X 0,Y 203.12,Z 446.247,A -85,B 0,C 180,E1 -21350.243,E2 -21350.243} C_VEL
LIN {X 0,Y 205.764,Z 441.154,A -85,B 0,C 180,E1 -21353.128,E2 -21353.128} C_VEL
LIN {X 0,Y 209.818,Z 433.77,A -85,B 0,C 180,E1 -21356.348,E2 -21356.348} C_VEL
LIN {X 0,Y 213.971,Z 425.922,A -85,B 0,C 180,E1 -21358.978,E2 -21358.978} C_VEL
LIN {X 0,Y 216.343,Z 419.881,A -85,B 0,C 180,E1 -21360.774,E2 -21360.774} C_VEL
LIN {X 0,Y 218.707,Z 410.597,A -85,B 0,C 180,E1 -21363.332,E2 -21363.332} C_VEL
LIN {X 0,Y 220.029,Z 401.683,A -85,B 0,C 180,E1 -21365.647,E2 -21365.647} C_VEL
LIN {X 0,Y 220.538,Z 392.574,A -85,B 0,C 180,E1 -21367.928,E2 -21367.928} C_VEL
LIN {X 0,Y 220.224,Z 382.305,A -85,B 0,C 180,E1 -21370.554,E2 -21370.554} C_VEL
LIN {X 0,Y 219.484,Z 376.013,A -85,B 0,C 180,E1 -21372.256,E2 -21372.256} C_VEL
LIN {X 0,Y 218.226,Z 371.826,A -85,B 0,C 180,E1 -21373.713,E2 -21373.713} C_VEL
LIN {X 0,Y 217.138,Z 368.474,A -85,B 0,C 180,E1 -21374.957,E2 -21374.957} C_VEL
LIN {X 0,Y 214.789,Z 363.249,A -85,B 0,C 180,E1 -21377.309,E2 -21377.309} C_VEL
LIN {X 0,Y 214.318,Z 361.859,A -85,B 0,C 180,E1 -21377.901,E2 -21377.901} C_VEL
LIN {X 0,Y 212.097,Z 358.132,A -85,B 0,C 180,E1 -21380.135,E2 -21380.135} C_VEL
LIN {X 0,Y 211.067,Z 354.926,A -85,B 0,C 180,E1 -21381.737,E2 -21381.737} C_VEL
LIN {X 0,Y 207.773,Z 349.495,A -85,B 0,C 180,E1 -21386.56,E2 -21386.56} C_VEL
LIN {X 0,Y 206.873,Z 346.305,A -85,B 0,C 180,E1 -21389.363,E2 -21389.363} C_VEL
LIN {X 0,Y 205.955,Z 344.131,A -85,B 0,C 180,E1 -21394.751,E2 -21394.751} C_VEL
LIN {X 0,Y 206.531,Z 343.513,A -85,B 0,C 180,E1 -21398.018,E2 -21398.018} C_VEL
LIN {X 0,Y 209.166,Z 346.509,A -85,B 0,C 180,E1 -21404.407,E2 -21404.407} C_VEL
LIN {X 0,Y 210.246,Z 347.032,A -85,B 0,C 180,E1 -21405.79,E2 -21405.79} C_VEL
LIN {X 0,Y 212.199,Z 350.174,A -85,B 0,C 180,E1 -21408.538,E2 -21408.538} C_VEL
LIN {X 0,Y 213.908,Z 351.744,A -85,B 0,C 180,E1 -21410.287,E2 -21410.287} C_VEL
LIN {X 0,Y 218.66,Z 359.467,A -85,B 0,C 180,E1 -21415.128,E2 -21415.128} C_VEL
LIN {X 0,Y 221.26,Z 364.636,A -85,B 0,C 180,E1 -21417.731,E2 -21417.731} C_VEL
LIN {X 0,Y 224.027,Z 372.73,A -85,B 0,C 180,E1 -21421.04,E2 -21421.04} C_VEL
LIN {X 0,Y 225.184,Z 377.723,A -85,B 0,C 180,E1 -21422.885,E2 -21422.885} C_VEL
LIN {X 0,Y 225.832,Z 385.001,A -85,B 0,C 180,E1 -21425.357,E2 -21425.357} C_VEL
LIN {X 0,Y 225.791,Z 386.354,A -85,B 0,C 180,E1 -21425.806,E2 -21425.806} C_VEL
LIN {X 0,Y 221.781,Z 395.617,A -85,B 0,C 180,E1 -21427.984,E2 -21427.984} C_VEL
LIN {X 0,Y 217.926,Z 403.291,A -85,B 0,C 180,E1 -21430.217,E2 -21430.217} C_VEL
LIN {X 0,Y 213.843,Z 410.553,A -85,B 0,C 180,E1 -21432.898,E2 -21432.898} C_VEL
LIN {X 0,Y 210.492,Z 416.009,A -85,B 0,C 180,E1 -21435.492,E2 -21435.492} C_VEL
LIN {X 0,Y 206.614,Z 421.645,A -85,B 0,C 180,E1 -21439.049,E2 -21439.049} C_VEL
LIN {X 0,Y 203.81,Z 425.259,A -85,B 0,C 180,E1 -21442.291,E2 -21442.291} C_VEL
LIN {X 0,Y 201.836,Z 427.379,A -85,B 0,C 180,E1 -21445.131,E2 -21445.131} C_VEL
LIN {X 0,Y 200.024,Z 428.832,A -85,B 0,C 180,E1 -21448.55,E2 -21448.55} C_VEL
LIN {X 0,Y 198.73,Z 429.154,A -85,B 0,C 180,E1 -21452.037,E2 -21452.037} C_VEL
LIN {X 0,Y 198.019,Z 428.409,A -85,B 0,C 180,E1 -21455.283,E2 -21455.283} C_VEL
LIN {X 0,Y 197.731,Z 426.648,A -85,B 0,C 180,E1 -21458.56,E2 -21458.56} C_VEL
LIN {X 0,Y 197.947,Z 423.197,A -85,B 0,C 180,E1 -21462.422,E2 -21462.422} C_VEL
LIN {X 0,Y 198.551,Z 418.892,A -85,B 0,C 180,E1 -21465.789,E2 -21465.789} C_VEL
LIN {X 0,Y 199.552,Z 413.096,A -85,B 0,C 180,E1 -21469.217,E2 -21469.217} C_VEL
LIN {X 0,Y 200.601,Z 407.059,A -85,B 0,C 180,E1 -21472.036,E2 -21472.036} C_VEL
LIN {X 0,Y 202.179,Z 399.156,A -85,B 0,C 180,E1 -21474.999,E2 -21474.999} C_VEL
LIN {X 0,Y 203.995,Z 390.085,A -85,B 0,C 180,E1 -21477.724,E2 -21477.724} C_VEL
LIN {X 0,Y 205.847,Z 380.564,A -85,B 0,C 180,E1 -21480.044,E2 -21480.044} C_VEL
LIN {X 0,Y 207.92,Z 368.92,A -85,B 0,C 180,E1 -21482.304,E2 -21482.304} C_VEL
LIN {X 0,Y 208.719,Z 363.258,A -85,B 0,C 180,E1 -21483.233,E2 -21483.233} C_VEL
LIN {X 0,Y 206.659,Z 352.693,A -85,B 0,C 180,E1 -21485.027,E2 -21485.027} C_VEL
LIN {X 0,Y 203.278,Z 340.848,A -85,B 0,C 180,E1 -21486.795,E2 -21486.795} C_VEL
LIN {X 0,Y 199.586,Z 329.624,A -85,B 0,C 180,E1 -21488.233,E2 -21488.233} C_VEL
LIN {X 0,Y 199.73,Z 329.606,A -85,B 0,C 180,E1 -21491.816,E2 -21491.816} C_VEL
LIN {X 0,Y 199.817,Z 329.596,A -85,B 0,C 180,E1 -21495.747,E2 -21495.747} C_VEL
LIN {X 0,Y 200.023,Z 329.571,A -85,B 0,C 180,E1 -21499.882,E2 -21499.882} C_VEL
LIN {X 0,Y 200.015,Z 329.567,A -85,B 0,C 180,E1 -21503.949,E2 -21503.949} C_VEL
LIN {X 0,Y 200.32,Z 329.532,A -85,B 0,C 180,E1 -21507.989,E2 -21507.989} C_VEL
LIN {X 0,Y 200.48,Z 329.508,A -85,B 0,C 180,E1 -21510,E2 -21510} C_VEL
LIN {X 0,Y 200.024,Z 329.568,A -85,B 0,C 180,E1 -21514.03,E2 -21514.03} C_VEL
LIN {X 0,Y 200.079,Z 329.56,A -85,B 0,C 180,E1 -21518.077,E2 -21518.077} C_VEL
LIN {X 0,Y 199.876,Z 329.588,A -85,B 0,C 180,E1 -21522.179,E2 -21522.179} C_VEL
LIN {X 0,Y 199.806,Z 329.596,A -85,B 0,C 180,E1 -21526.343,E2 -21526.343} C_VEL
LIN {X 0,Y 199.701,Z 329.607,A -85,B 0,C 180,E1 -21530.605,E2 -21530.605} C_VEL
LIN {X 0,Y 199.674,Z 329.611,A -85,B 0,C 180,E1 -21534.984,E2 -21534.984} C_VEL
LIN {X 0,Y 199.676,Z 329.609,A -85,B 0,C 180,E1 -21539.522,E2 -21539.522} C_VEL
LIN {X 0,Y 199.665,Z 329.614,A -85,B 0,C 180,E1 -21542.352,E2 -21542.352} C_VEL
LIN {X 0,Y 199.641,Z 329.614,A -85,B 0,C 180,E1 -21546.76,E2 -21546.76} C_VEL
LIN {X 0,Y 199.64,Z 329.612,A -85,B 0,C 180,E1 -21549.321,E2 -21549.321} C_VEL
LIN {X 0,Y 199.581,Z 329.622,A -85,B 0,C 180,E1 -21554.771,E2 -21554.771} C_VEL
LIN {X 0,Y 199.581,Z 329.624,A -85,B 0,C 180,E1 -21558.006,E2 -21558.006} C_VEL
LIN {X 0,Y 199.612,Z 329.619,A -85,B 0,C 180,E1 -21560.768,E2 -21560.768} C_VEL
LIN {X 0,Y 199.626,Z 329.617,A -85,B 0,C 180,E1 -21565.716,E2 -21565.716} C_VEL
LIN {X 0,Y 199.705,Z 329.608,A -85,B 0,C 180,E1 -21568.138,E2 -21568.138} C_VEL
LIN {X 0,Y 199.688,Z 329.607,A -85,B 0,C 180,E1 -21572.772,E2 -21572.772} C_VEL
LIN {X 0,Y 199.715,Z 329.609,A -85,B 0,C 180,E1 -21577.227,E2 -21577.227} C_VEL
LIN {X 0,Y 199.797,Z 329.594,A -85,B 0,C 180,E1 -21581.76,E2 -21581.76} C_VEL
LIN {X 0,Y 199.822,Z 329.593,A -85,B 0,C 180,E1 -21585.748,E2 -21585.748} C_VEL
LIN {X 0,Y 200.025,Z 329.565,A -85,B 0,C 180,E1 -21589.882,E2 -21589.882} C_VEL
LIN {X 0,Y 200.022,Z 329.568,A -85,B 0,C 180,E1 -21593.95,E2 -21593.95} C_VEL
LIN {X 0,Y 200.322,Z 329.527,A -85,B 0,C 180,E1 -21597.99,E2 -21597.99} C_VEL
LIN {X 0,Y 200.479,Z 329.51,A -85,B 0,C 180,E1 -21600,E2 -21600} C_VEL
LIN {X 0,Y 200.014,Z 329.568,A -85,B 0,C 180,E1 -21604.03,E2 -21604.03} C_VEL
LIN {X 0,Y 200.084,Z 329.559,A -85,B 0,C 180,E1 -21608.077,E2 -21608.077} C_VEL
LIN {X 0,Y 199.873,Z 329.587,A -85,B 0,C 180,E1 -21612.18,E2 -21612.18} C_VEL
LIN {X 0,Y 199.792,Z 329.597,A -85,B 0,C 180,E1 -21616.345,E2 -21616.345} C_VEL
LIN {X 0,Y 199.677,Z 329.61,A -85,B 0,C 180,E1 -21620.608,E2 -21620.608} C_VEL
LIN {X 0,Y 199.653,Z 329.601,A -85,B 0,C 180,E1 -21624.987,E2 -21624.987} C_VEL
LIN {X 0,Y 199.612,Z 329.613,A -85,B 0,C 180,E1 -21629.533,E2 -21629.533} C_VEL
LIN {X 0,Y 199.654,Z 329.617,A -85,B 0,C 180,E1 -21632.346,E2 -21632.346} C_VEL
LIN {X 0,Y 199.662,Z 329.614,A -85,B 0,C 180,E1 -21636.755,E2 -21636.755} C_VEL
LIN {X 0,Y 199.741,Z 329.617,A -85,B 0,C 180,E1 -21638.327,E2 -21638.327} C_VEL
LIN {X 0,Y 200.485,Z 333.686,A -85,B 0,C 180,E1 -21642.595,E2 -21642.595} C_VEL
LIN {X 0,Y 201.34,Z 338.288,A -85,B 0,C 180,E1 -21647.142,E2 -21647.142} C_VEL
LIN {X 0,Y 202.111,Z 342.65,A -85,B 0,C 180,E1 -21651.25,E2 -21651.25} C_VEL
LIN {X 0,Y 201.831,Z 345.378,A -85,B 0,C 180,E1 -21653.703,E2 -21653.703} C_VEL
LIN {X 0,Y 200.428,Z 350.638,A -85,B 0,C 180,E1 -21658.266,E2 -21658.266} C_VEL
LIN {X 0,Y 200.13,Z 351.846,A -85,B 0,C 180,E1 -21659.309,E2 -21659.309} C_VEL
LIN {X 0,Y 201.774,Z 366.009,A -85,B 0,C 180,E1 -21660.55,E2 -21660.55} C_VEL
LIN {X 0,Y 202.999,Z 379.47,A -85,B 0,C 180,E1 -21662.138,E2 -21662.138} C_VEL
LIN {X 0,Y 203.781,Z 391.708,A -85,B 0,C 180,E1 -21663.943,E2 -21663.943} C_VEL
LIN {X 0,Y 204.136,Z 403.743,A -85,B 0,C 180,E1 -21666.138,E2 -21666.138} C_VEL
LIN {X 0,Y 204.052,Z 411.226,A -85,B 0,C 180,E1 -21667.737,E2 -21667.737} C_VEL
LIN {X 0,Y 201.889,Z 421.813,A -85,B 0,C 180,E1 -21670.4,E2 -21670.4} C_VEL
LIN {X 0,Y 200.271,Z 430.594,A -85,B 0,C 180,E1 -21673.171,E2 -21673.171} C_VEL
LIN {X 0,Y 198.976,Z 438.23,A -85,B 0,C 180,E1 -21676.207,E2 -21676.207} C_VEL
LIN {X 0,Y 198.201,Z 444.533,A -85,B 0,C 180,E1 -21679.375,E2 -21679.375} C_VEL
LIN {X 0,Y 197.317,Z 447.042,A -85,B 0,C 180,E1 -21680.906,E2 -21680.906} C_VEL
LIN {X 0,Y 194.267,Z 450.432,A -85,B 0,C 180,E1 -21683.489,E2 -21683.489} C_VEL
LIN {X 0,Y 191.858,Z 452.545,A -85,B 0,C 180,E1 -21685.668,E2 -21685.668} C_VEL
LIN {X 0,Y 190.933,Z 453.852,A -85,B 0,C 180,E1 -21687.389,E2 -21687.389} C_VEL
LIN {X 0,Y 190.909,Z 454.239,A -85,B 0,C 180,E1 -21687.975,E2 -21687.975} C_VEL
LIN {X 0,Y 191.246,Z 455.533,A -85,B 0,C 180,E1 -21690,E2 -21690} C_VEL
LIN {X 0,Y 190.659,Z 456.785,A -85,B 0,C 180,E1 -21694.228,E2 -21694.228} C_VEL
LIN {X 0,Y 190.557,Z 456.492,A -85,B 0,C 180,E1 -21698.484,E2 -21698.484} C_VEL
LIN {X 0,Y 191.36,Z 454.635,A -85,B 0,C 180,E1 -21702.73,E2 -21702.73} C_VEL
LIN {X 0,Y 193.354,Z 451.287,A -85,B 0,C 180,E1 -21706.905,E2 -21706.905} C_VEL
LIN {X 0,Y 195.552,Z 447.686,A -85,B 0,C 180,E1 -21709.964,E2 -21709.964} C_VEL
LIN {X 0,Y 198.228,Z 443.119,A -85,B 0,C 180,E1 -21712.954,E2 -21712.954} C_VEL
LIN {X 0,Y 202.161,Z 436.461,A -85,B 0,C 180,E1 -21716.311,E2 -21716.311} C_VEL
LIN {X 0,Y 206.347,Z 429.332,A -85,B 0,C 180,E1 -21719.035,E2 -21719.035} C_VEL
LIN {X 0,Y 209.19,Z 423.76,A -85,B 0,C 180,E1 -21720.82,E2 -21720.82} C_VEL
LIN {X 0,Y 211.971,Z 415.373,A -85,B 0,C 180,E1 -21723.384,E2 -21723.384} C_VEL
LIN {X 0,Y 213.792,Z 407.174,A -85,B 0,C 180,E1 -21725.697,E2 -21725.697} C_VEL
LIN {X 0,Y 215.009,Z 397.21,A -85,B 0,C 180,E1 -21728.393,E2 -21728.393} C_VEL
LIN {X 0,Y 215.265,Z 387.367,A -85,B 0,C 180,E1 -21731.074,E2 -21731.074} C_VEL
LIN {X 0,Y 214.888,Z 380.479,A -85,B 0,C 180,E1 -21733.051,E2 -21733.051} C_VEL
LIN {X 0,Y 213.988,Z 376.945,A -85,B 0,C 180,E1 -21734.359,E2 -21734.359} C_VEL
LIN {X 0,Y 212.645,Z 372.897,A -85,B 0,C 180,E1 -21736.047,E2 -21736.047} C_VEL
LIN {X 0,Y 210.971,Z 368.255,A -85,B 0,C 180,E1 -21738.221,E2 -21738.221} C_VEL
LIN {X 0,Y 208.948,Z 364.164,A -85,B 0,C 180,E1 -21740.68,E2 -21740.68} C_VEL
LIN {X 0,Y 207.898,Z 360.891,A -85,B 0,C 180,E1 -21742.519,E2 -21742.519} C_VEL
LIN {X 0,Y 205.039,Z 354.85,A -85,B 0,C 180,E1 -21747.947,E2 -21747.947} C_VEL
LIN {X 0,Y 204.846,Z 353.509,A -85,B 0,C 180,E1 -21749.062,E2 -21749.062} C_VEL
LIN {X 0,Y 204.252,Z 352.205,A -85,B 0,C 180,E1 -21751.202,E2 -21751.202} C_VEL
LIN {X 0,Y 204.012,Z 350.738,A -85,B 0,C 180,E1 -21755.582,E2 -21755.582} C_VEL
LIN {X 0,Y 204.488,Z 350.343,A -85,B 0,C 180,E1 -21758.12,E2 -21758.12} C_VEL
LIN {X 0,Y 206.672,Z 353.14,A -85,B 0,C 180,E1 -21764.214,E2 -21764.214} C_VEL
LIN {X 0,Y 207.966,Z 354.47,A -85,B 0,C 180,E1 -21766.316,E2 -21766.316} C_VEL
LIN {X 0,Y 210.997,Z 358.717,A -85,B 0,C 180,E1 -21770.413,E2 -21770.413} C_VEL
LIN {X 0,Y 214.339,Z 364.572,A -85,B 0,C 180,E1 -21774.355,E2 -21774.355} C_VEL
LIN {X 0,Y 216.812,Z 369.797,A -85,B 0,C 180,E1 -21777.213,E2 -21777.213} C_VEL
LIN {X 0,Y 219.236,Z 378.279,A -85,B 0,C 180,E1 -21780.918,E2 -21780.918} C_VEL
LIN {X 0,Y 219.93,Z 382.964,A -85,B 0,C 180,E1 -21782.747,E2 -21782.747} C_VEL
LIN {X 0,Y 220.127,Z 388.016,A -85,B 0,C 180,E1 -21784.579,E2 -21784.579} C_VEL
LIN {X 0,Y 219.765,Z 389.757,A -85,B 0,C 180,E1 -21785.092,E2 -21785.092} C_VEL
LIN {X 0,Y 215.069,Z 399.235,A -85,B 0,C 180,E1 -21787.51,E2 -21787.51} C_VEL
LIN {X 0,Y 210.676,Z 407.129,A -85,B 0,C 180,E1 -21790.086,E2 -21790.086} C_VEL
LIN {X 0,Y 206.615,Z 413.616,A -85,B 0,C 180,E1 -21792.772,E2 -21792.772} C_VEL
LIN {X 0,Y 202.437,Z 419.647,A -85,B 0,C 180,E1 -21796.125,E2 -21796.125} C_VEL
LIN {X 0,Y 198.857,Z 424.192,A -85,B 0,C 180,E1 -21799.618,E2 -21799.618} C_VEL
LIN {X 0,Y 195.939,Z 427.364,A -85,B 0,C 180,E1 -21803.238,E2 -21803.238} C_VEL
LIN {X 0,Y 194.339,Z 428.721,A -85,B 0,C 180,E1 -21805.719,E2 -21805.719} C_VEL
LIN {X 0,Y 192.727,Z 429.643,A -85,B 0,C 180,E1 -21808.932,E2 -21808.932} C_VEL
LIN {X 0,Y 191.512,Z 429.597,A -85,B 0,C 180,E1 -21812.43,E2 -21812.43} C_VEL
LIN {X 0,Y 190.816,Z 428.403,A -85,B 0,C 180,E1 -21816.107,E2 -21816.107} C_VEL
LIN {X 0,Y 190.623,Z 426.423,A -85,B 0,C 180,E1 -21819.263,E2 -21819.263} C_VEL
LIN {X 0,Y 190.887,Z 423.344,A -85,B 0,C 180,E1 -21822.578,E2 -21822.578} C_VEL
LIN {X 0,Y 191.578,Z 418.456,A -85,B 0,C 180,E1 -21826.38,E2 -21826.38} C_VEL
LIN {X 0,Y 192.659,Z 412.173,A -85,B 0,C 180,E1 -21830.001,E2 -21830.001} C_VEL
LIN {X 0,Y 194.103,Z 404.703,A -85,B 0,C 180,E1 -21833.363,E2 -21833.363} C_VEL
LIN {X 0,Y 195.674,Z 396.921,A -85,B 0,C 180,E1 -21836.171,E2 -21836.171} C_VEL
LIN {X 0,Y 197.754,Z 387.059,A -85,B 0,C 180,E1 -21839.012,E2 -21839.012} C_VEL
LIN {X 0,Y 199.851,Z 376.107,A -85,B 0,C 180,E1 -21841.54,E2 -21841.54} C_VEL
LIN {X 0,Y 201.837,Z 364.501,A -85,B 0,C 180,E1 -21843.643,E2 -21843.643} C_VEL
LIN {X 0,Y 200.04,Z 354.959,A -85,B 0,C 180,E1 -21845.342,E2 -21845.342} C_VEL
LIN {X 0,Y 196.859,Z 343.546,A -85,B 0,C 180,E1 -21847.154,E2 -21847.154} C_VEL
LIN {X 0,Y 192.553,Z 330.501,A -85,B 0,C 180,E1 -21848.943,E2 -21848.943} C_VEL
LIN {X 0,Y 192.712,Z 330.48,A -85,B 0,C 180,E1 -21853.037,E2 -21853.037} C_VEL
LIN {X 0,Y 192.795,Z 330.472,A -85,B 0,C 180,E1 -21857.366,E2 -21857.366} C_VEL
LIN {X 0,Y 193.029,Z 330.443,A -85,B 0,C 180,E1 -21861.626,E2 -21861.626} C_VEL
LIN {X 0,Y 193.262,Z 330.411,A -85,B 0,C 180,E1 -21867.916,E2 -21867.916} C_VEL
LIN {X 0,Y 193.444,Z 330.384,A -85,B 0,C 180,E1 -21870,E2 -21870} C_VEL
LIN {X 0,Y 192.969,Z 330.447,A -85,B 0,C 180,E1 -21874.177,E2 -21874.177} C_VEL
LIN {X 0,Y 193.029,Z 330.439,A -85,B 0,C 180,E1 -21878.374,E2 -21878.374} C_VEL
LIN {X 0,Y 192.803,Z 330.468,A -85,B 0,C 180,E1 -21882.633,E2 -21882.633} C_VEL
LIN {X 0,Y 192.759,Z 330.473,A -85,B 0,C 180,E1 -21886.959,E2 -21886.959} C_VEL
LIN {X 0,Y 192.638,Z 330.485,A -85,B 0,C 180,E1 -21891.397,E2 -21891.397} C_VEL
LIN {X 0,Y 192.665,Z 330.485,A -85,B 0,C 180,E1 -21894.225,E2 -21894.225} C_VEL
LIN {X 0,Y 192.651,Z 330.484,A -85,B 0,C 180,E1 -21898.892,E2 -21898.892} C_VEL
LIN {X 0,Y 192.601,Z 330.492,A -85,B 0,C 180,E1 -21903.186,E2 -21903.186} C_VEL
LIN {X 0,Y 192.61,Z 330.49,A -85,B 0,C 180,E1 -21906.608,E2 -21906.608} C_VEL
LIN {X 0,Y 192.525,Z 330.501,A -85,B 0,C 180,E1 -21911.078,E2 -21911.078} C_VEL
LIN {X 0,Y 192.493,Z 330.503,A -85,B 0,C 180,E1 -21916.077,E2 -21916.077} C_VEL
LIN {X 0,Y 192.52,Z 330.504,A -85,B 0,C 180,E1 -21920.051,E2 -21920.051} C_VEL
LIN {X 0,Y 192.578,Z 330.492,A -85,B 0,C 180,E1 -21924.274,E2 -21924.274} C_VEL
LIN {X 0,Y 192.609,Z 330.493,A -85,B 0,C 180,E1 -21929.281,E2 -21929.281} C_VEL
LIN {X 0,Y 192.667,Z 330.483,A -85,B 0,C 180,E1 -21931.692,E2 -21931.692} C_VEL
LIN {X 0,Y 192.687,Z 330.481,A -85,B 0,C 180,E1 -21936.346,E2 -21936.346} C_VEL
LIN {X 0,Y 192.732,Z 330.475,A -85,B 0,C 180,E1 -21941.46,E2 -21941.46} C_VEL
LIN {X 0,Y 192.751,Z 330.477,A -85,B 0,C 180,E1 -21945.213,E2 -21945.213} C_VEL
LIN {X 0,Y 192.947,Z 330.447,A -85,B 0,C 180,E1 -21949.567,E2 -21949.567} C_VEL
LIN {X 0,Y 192.985,Z 330.445,A -85,B 0,C 180,E1 -21953.728,E2 -21953.728} C_VEL
LIN {X 0,Y 193.264,Z 330.406,A -85,B 0,C 180,E1 -21957.916,E2 -21957.916} C_VEL
LIN {X 0,Y 193.443,Z 330.387,A -85,B 0,C 180,E1 -21960,E2 -21960} C_VEL
LIN {X 0,Y 192.96,Z 330.447,A -85,B 0,C 180,E1 -21964.178,E2 -21964.178} C_VEL
LIN {X 0,Y 193.033,Z 330.439,A -85,B 0,C 180,E1 -21968.374,E2 -21968.374} C_VEL
LIN {X 0,Y 192.8,Z 330.467,A -85,B 0,C 180,E1 -21972.634,E2 -21972.634} C_VEL
LIN {X 0,Y 192.75,Z 330.475,A -85,B 0,C 180,E1 -21976.96,E2 -21976.96} C_VEL
LIN {X 0,Y 192.612,Z 330.488,A -85,B 0,C 180,E1 -21981.4,E2 -21981.4} C_VEL
LIN {X 0,Y 192.642,Z 330.477,A -85,B 0,C 180,E1 -21984.208,E2 -21984.208} C_VEL
LIN {X 0,Y 192.605,Z 330.486,A -85,B 0,C 180,E1 -21988.866,E2 -21988.866} C_VEL
LIN {X 0,Y 192.598,Z 330.494,A -85,B 0,C 180,E1 -21993.186,E2 -21993.186} C_VEL
LIN {X 0,Y 192.684,Z 330.502,A -85,B 0,C 180,E1 -21998.08,E2 -21998.08} C_VEL
LIN {X 0,Y 193.582,Z 335.495,A -85,B 0,C 180,E1 -22003.439,E2 -22003.439} C_VEL
LIN {X 0,Y 194.431,Z 339.805,A -85,B 0,C 180,E1 -22007.816,E2 -22007.816} C_VEL
LIN {X 0,Y 194.98,Z 342.94,A -85,B 0,C 180,E1 -22010.892,E2 -22010.892} C_VEL
LIN {X 0,Y 195.01,Z 344.593,A -85,B 0,C 180,E1 -22012.454,E2 -22012.454} C_VEL
LIN {X 0,Y 193.691,Z 349.658,A -85,B 0,C 180,E1 -22017.025,E2 -22017.025} C_VEL
LIN {X 0,Y 193.228,Z 351.373,A -85,B 0,C 180,E1 -22018.564,E2 -22018.564} C_VEL
LIN {X 0,Y 194.74,Z 364.651,A -85,B 0,C 180,E1 -22019.767,E2 -22019.767} C_VEL
LIN {X 0,Y 195.905,Z 377.327,A -85,B 0,C 180,E1 -22021.272,E2 -22021.272} C_VEL
LIN {X 0,Y 196.747,Z 390.564,A -85,B 0,C 180,E1 -22023.256,E2 -22023.256} C_VEL
LIN {X 0,Y 197.112,Z 401.293,A -85,B 0,C 180,E1 -22025.232,E2 -22025.232} C_VEL
LIN {X 0,Y 197.177,Z 410.372,A -85,B 0,C 180,E1 -22027.221,E2 -22027.221} C_VEL
LIN {X 0,Y 195.059,Z 420.617,A -85,B 0,C 180,E1 -22029.858,E2 -22029.858} C_VEL
LIN {X 0,Y 193.426,Z 429.032,A -85,B 0,C 180,E1 -22032.557,E2 -22032.557} C_VEL
LIN {X 0,Y 192.066,Z 436.901,A -85,B 0,C 180,E1 -22035.7,E2 -22035.7} C_VEL
LIN {X 0,Y 191.301,Z 442.21,A -85,B 0,C 180,E1 -22038.343,E2 -22038.343} C_VEL
LIN {X 0,Y 190.899,Z 447.391,A -85,B 0,C 180,E1 -22041.532,E2 -22041.532} C_VEL
LIN {X 0,Y 190.842,Z 450.407,A -85,B 0,C 180,E1 -22043.887,E2 -22043.887} C_VEL
LIN {X 0,Y 190.853,Z 452.394,A -85,B 0,C 180,E1 -22045.776,E2 -22045.776} C_VEL
LIN {X 0,Y 190.909,Z 454.239,A -85,B 0,C 180,E1 -22047.975,E2 -22047.975} C_VEL
LIN {X 0,Y 190.287,Z 454.927,A -85,B 0,C 180,E1 -22049.128,E2 -22049.128} C_VEL
LIN {X 0,Y 187.357,Z 455.538,A -85,B 0,C 180,E1 -22050.948,E2 -22050.948} C_VEL
LIN {X 0,Y 184.32,Z 455.889,A -85,B 0,C 180,E1 -22052.835,E2 -22052.835} C_VEL
LIN {X 0,Y 183.591,Z 456.066,A -85,B 0,C 180,E1 -22054.069,E2 -22054.069} C_VEL
LIN {X 0,Y 183.41,Z 456.237,A -85,B 0,C 180,E1 -22056.601,E2 -22056.601} C_VEL
LIN {X 0,Y 183.817,Z 455.336,A -85,B 0,C 180,E1 -22061.021,E2 -22061.021} C_VEL
LIN {X 0,Y 185.287,Z 452.891,A -85,B 0,C 180,E1 -22065.398,E2 -22065.398} C_VEL
LIN {X 0,Y 187.988,Z 448.931,A -85,B 0,C 180,E1 -22069.662,E2 -22069.662} C_VEL
LIN {X 0,Y 191.005,Z 444.39,A -85,B 0,C 180,E1 -22073.091,E2 -22073.091} C_VEL
LIN {X 0,Y 193.927,Z 439.777,A -85,B 0,C 180,E1 -22075.778,E2 -22075.778} C_VEL
LIN {X 0,Y 197.964,Z 433.529,A -85,B 0,C 180,E1 -22078.638,E2 -22078.638} C_VEL
LIN {X 0,Y 202.466,Z 426.016,A -85,B 0,C 180,E1 -22081.378,E2 -22081.378} C_VEL
LIN {X 0,Y 205.306,Z 419.036,A -85,B 0,C 180,E1 -22083.677,E2 -22083.677} C_VEL
LIN {X 0,Y 207.734,Z 410.419,A -85,B 0,C 180,E1 -22086.302,E2 -22086.302} C_VEL
LIN {X 0,Y 209.441,Z 400.881,A -85,B 0,C 180,E1 -22089.096,E2 -22089.096} C_VEL
LIN {X 0,Y 210.179,Z 391.003,A -85,B 0,C 180,E1 -22091.972,E2 -22091.972} C_VEL
LIN {X 0,Y 210.121,Z 384.425,A -85,B 0,C 180,E1 -22094.019,E2 -22094.019} C_VEL
LIN {X 0,Y 208.933,Z 379.434,A -85,B 0,C 180,E1 -22096.076,E2 -22096.076} C_VEL
LIN {X 0,Y 207.271,Z 374.311,A -85,B 0,C 180,E1 -22098.607,E2 -22098.607} C_VEL
LIN {X 0,Y 204.747,Z 367.158,A -85,B 0,C 180,E1 -22102.904,E2 -22102.904} C_VEL
LIN {X 0,Y 202.344,Z 360.985,A -85,B 0,C 180,E1 -22108.601,E2 -22108.601} C_VEL
LIN {X 0,Y 201.889,Z 359.165,A -85,B 0,C 180,E1 -22110.833,E2 -22110.833} C_VEL
LIN {X 0,Y 201.563,Z 357.524,A -85,B 0,C 180,E1 -22115.265,E2 -22115.265} C_VEL
LIN {X 0,Y 201.933,Z 357.07,A -85,B 0,C 180,E1 -22117.49,E2 -22117.49} C_VEL
LIN {X 0,Y 204.127,Z 359.955,A -85,B 0,C 180,E1 -22124.588,E2 -22124.588} C_VEL
LIN {X 0,Y 204.985,Z 360.914,A -85,B 0,C 180,E1 -22126.113,E2 -22126.113} C_VEL
LIN {X 0,Y 207.622,Z 365.01,A -85,B 0,C 180,E1 -22130.256,E2 -22130.256} C_VEL
LIN {X 0,Y 210.482,Z 370.634,A -85,B 0,C 180,E1 -22134.251,E2 -22134.251} C_VEL
LIN {X 0,Y 211.917,Z 373.922,A -85,B 0,C 180,E1 -22136.197,E2 -22136.197} C_VEL
LIN {X 0,Y 213.608,Z 380.533,A -85,B 0,C 180,E1 -22139.413,E2 -22139.413} C_VEL
LIN {X 0,Y 214.353,Z 384.463,A -85,B 0,C 180,E1 -22141.174,E2 -22141.174} C_VEL
LIN {X 0,Y 214.427,Z 390.979,A -85,B 0,C 180,E1 -22143.758,E2 -22143.758} C_VEL
LIN {X 0,Y 212.278,Z 395.661,A -85,B 0,C 180,E1 -22144.979,E2 -22144.979} C_VEL
LIN {X 0,Y 207.873,Z 403.58,A -85,B 0,C 180,E1 -22147.284,E2 -22147.284} C_VEL
LIN {X 0,Y 203.361,Z 410.791,A -85,B 0,C 180,E1 -22149.95,E2 -22149.95} C_VEL
LIN {X 0,Y 199.277,Z 416.628,A -85,B 0,C 180,E1 -22152.734,E2 -22152.734} C_VEL
LIN {X 0,Y 195.502,Z 421.531,A -85,B 0,C 180,E1 -22155.779,E2 -22155.779} C_VEL
LIN {X 0,Y 191.978,Z 425.547,A -85,B 0,C 180,E1 -22159.237,E2 -22159.237} C_VEL
LIN {X 0,Y 189.594,Z 427.868,A -85,B 0,C 180,E1 -22162.07,E2 -22162.07} C_VEL
LIN {X 0,Y 187.194,Z 429.682,A -85,B 0,C 180,E1 -22165.702,E2 -22165.702} C_VEL
LIN {X 0,Y 185.378,Z 430.351,A -85,B 0,C 180,E1 -22169.528,E2 -22169.528} C_VEL
LIN {X 0,Y 184.288,Z 429.944,A -85,B 0,C 180,E1 -22172.965,E2 -22172.965} C_VEL
LIN {X 0,Y 183.676,Z 428.506,A -85,B 0,C 180,E1 -22176.532,E2 -22176.532} C_VEL
LIN {X 0,Y 183.581,Z 425.579,A -85,B 0,C 180,E1 -22180.602,E2 -22180.602} C_VEL
LIN {X 0,Y 184.151,Z 420.895,A -85,B 0,C 180,E1 -22184.913,E2 -22184.913} C_VEL
LIN {X 0,Y 185.111,Z 415.282,A -85,B 0,C 180,E1 -22188.633,E2 -22188.633} C_VEL
LIN {X 0,Y 186.443,Z 408.057,A -85,B 0,C 180,E1 -22192.335,E2 -22192.335} C_VEL
LIN {X 0,Y 188.005,Z 400.658,A -85,B 0,C 180,E1 -22195.326,E2 -22195.326} C_VEL
LIN {X 0,Y 189.93,Z 391.426,A -85,B 0,C 180,E1 -22198.328,E2 -22198.328} C_VEL
LIN {X 0,Y 192.169,Z 380.731,A -85,B 0,C 180,E1 -22201.105,E2 -22201.105} C_VEL
LIN {X 0,Y 194.278,Z 369.46,A -85,B 0,C 180,E1 -22203.406,E2 -22203.406} C_VEL
LIN {X 0,Y 194.913,Z 365.66,A -85,B 0,C 180,E1 -22204.075,E2 -22204.075} C_VEL
LIN {X 0,Y 193.512,Z 357.594,A -85,B 0,C 180,E1 -22205.598,E2 -22205.598} C_VEL
LIN {X 0,Y 190.458,Z 346.368,A -85,B 0,C 180,E1 -22207.519,E2 -22207.519} C_VEL
LIN {X 0,Y 186.457,Z 334.366,A -85,B 0,C 180,E1 -22209.307,E2 -22209.307} C_VEL
LIN {X 0,Y 185.522,Z 331.377,A -85,B 0,C 180,E1 -22209.704,E2 -22209.704} C_VEL
LIN {X 0,Y 185.648,Z 331.36,A -85,B 0,C 180,E1 -22212.371,E2 -22212.371} C_VEL
LIN {X 0,Y 185.72,Z 331.354,A -85,B 0,C 180,E1 -22216.876,E2 -22216.876} C_VEL
LIN {X 0,Y 185.977,Z 331.323,A -85,B 0,C 180,E1 -22221.306,E2 -22221.306} C_VEL
LIN {X 0,Y 186.205,Z 331.29,A -85,B 0,C 180,E1 -22227.837,E2 -22227.837} C_VEL
LIN {X 0,Y 186.408,Z 331.261,A -85,B 0,C 180,E1 -22230,E2 -22230} C_VEL
LIN {X 0,Y 185.916,Z 331.326,A -85,B 0,C 180,E1 -22234.336,E2 -22234.336} C_VEL
LIN {X 0,Y 185.977,Z 331.319,A -85,B 0,C 180,E1 -22238.694,E2 -22238.694} C_VEL
LIN {X 0,Y 185.73,Z 331.347,A -85,B 0,C 180,E1 -22243.123,E2 -22243.123} C_VEL
LIN {X 0,Y 185.691,Z 331.353,A -85,B 0,C 180,E1 -22247.625,E2 -22247.625} C_VEL
LIN {X 0,Y 185.598,Z 331.363,A -85,B 0,C 180,E1 -22252.251,E2 -22252.251} C_VEL
LIN {X 0,Y 185.564,Z 331.369,A -85,B 0,C 180,E1 -22257.032,E2 -22257.032} C_VEL
LIN {X 0,Y 185.58,Z 331.365,A -85,B 0,C 180,E1 -22259.493,E2 -22259.493} C_VEL
LIN {X 0,Y 185.52,Z 331.375,A -85,B 0,C 180,E1 -22264.628,E2 -22264.628} C_VEL
LIN {X 0,Y 185.545,Z 331.37,A -85,B 0,C 180,E1 -22267.304,E2 -22267.304} C_VEL
LIN {X 0,Y 185.486,Z 331.378,A -85,B 0,C 180,E1 -22270.73,E2 -22270.73} C_VEL
LIN {X 0,Y 185.462,Z 331.379,A -85,B 0,C 180,E1 -22276.055,E2 -22276.055} C_VEL
LIN {X 0,Y 185.47,Z 331.383,A -85,B 0,C 180,E1 -22279.896,E2 -22279.896} C_VEL
LIN {X 0,Y 185.504,Z 331.375,A -85,B 0,C 180,E1 -22282.713,E2 -22282.713} C_VEL
LIN {X 0,Y 185.546,Z 331.372,A -85,B 0,C 180,E1 -22287.976,E2 -22287.976} C_VEL
LIN {X 0,Y 185.584,Z 331.366,A -85,B 0,C 180,E1 -22290.576,E2 -22290.576} C_VEL
LIN {X 0,Y 185.582,Z 331.368,A -85,B 0,C 180,E1 -22295.382,E2 -22295.382} C_VEL
LIN {X 0,Y 185.674,Z 331.354,A -85,B 0,C 180,E1 -22301.136,E2 -22301.136} C_VEL
LIN {X 0,Y 185.684,Z 331.354,A -85,B 0,C 180,E1 -22304.637,E2 -22304.637} C_VEL
LIN {X 0,Y 185.891,Z 331.326,A -85,B 0,C 180,E1 -22309.418,E2 -22309.418} C_VEL
LIN {X 0,Y 185.948,Z 331.322,A -85,B 0,C 180,E1 -22313.49,E2 -22313.49} C_VEL
LIN {X 0,Y 186.208,Z 331.285,A -85,B 0,C 180,E1 -22317.837,E2 -22317.837} C_VEL
LIN {X 0,Y 186.406,Z 331.263,A -85,B 0,C 180,E1 -22320,E2 -22320} C_VEL
LIN {X 0,Y 185.907,Z 331.326,A -85,B 0,C 180,E1 -22324.336,E2 -22324.336} C_VEL
LIN {X 0,Y 185.981,Z 331.319,A -85,B 0,C 180,E1 -22328.694,E2 -22328.694} C_VEL
LIN {X 0,Y 185.726,Z 331.346,A -85,B 0,C 180,E1 -22333.123,E2 -22333.123} C_VEL
LIN {X 0,Y 185.687,Z 331.354,A -85,B 0,C 180,E1 -22337.626,E2 -22337.626} C_VEL
LIN {X 0,Y 185.574,Z 331.364,A -85,B 0,C 180,E1 -22342.255,E2 -22342.255} C_VEL
LIN {X 0,Y 185.579,Z 331.354,A -85,B 0,C 180,E1 -22344.646,E2 -22344.646} C_VEL
LIN {X 0,Y 185.546,Z 331.365,A -85,B 0,C 180,E1 -22349.499,E2 -22349.499} C_VEL
LIN {X 0,Y 185.523,Z 331.376,A -85,B 0,C 180,E1 -22354.627,E2 -22354.627} C_VEL
LIN {X 0,Y 185.662,Z 331.505,A -85,B 0,C 180,E1 -22357.96,E2 -22357.96} C_VEL
LIN {X 0,Y 186.447,Z 335.765,A -85,B 0,C 180,E1 -22362.727,E2 -22362.727} C_VEL
LIN {X 0,Y 187.514,Z 341.295,A -85,B 0,C 180,E1 -22368.556,E2 -22368.556} C_VEL
LIN {X 0,Y 187.945,Z 344.467,A -85,B 0,C 180,E1 -22371.746,E2 -22371.746} C_VEL
LIN {X 0,Y 187.334,Z 347.306,A -85,B 0,C 180,E1 -22374.444,E2 -22374.444} C_VEL
LIN {X 0,Y 186.341,Z 350.847,A -85,B 0,C 180,E1 -22377.769,E2 -22377.769} C_VEL
LIN {X 0,Y 187.861,Z 364.659,A -85,B 0,C 180,E1 -22379.085,E2 -22379.085} C_VEL
LIN {X 0,Y 189.028,Z 377.733,A -85,B 0,C 180,E1 -22380.733,E2 -22380.733} C_VEL
LIN {X 0,Y 189.764,Z 390.422,A -85,B 0,C 180,E1 -22382.73,E2 -22382.73} C_VEL
LIN {X 0,Y 190.112,Z 401.363,A -85,B 0,C 180,E1 -22384.841,E2 -22384.841} C_VEL
LIN {X 0,Y 190.158,Z 410.27,A -85,B 0,C 180,E1 -22386.878,E2 -22386.878} C_VEL
LIN {X 0,Y 188.079,Z 420.174,A -85,B 0,C 180,E1 -22389.54,E2 -22389.54} C_VEL
LIN {X 0,Y 186.342,Z 428.829,A -85,B 0,C 180,E1 -22392.439,E2 -22392.439} C_VEL
LIN {X 0,Y 184.975,Z 436.622,A -85,B 0,C 180,E1 -22395.702,E2 -22395.702} C_VEL
LIN {X 0,Y 184.133,Z 442.824,A -85,B 0,C 180,E1 -22398.998,E2 -22398.998} C_VEL
LIN {X 0,Y 183.787,Z 447.724,A -85,B 0,C 180,E1 -22402.308,E2 -22402.308} C_VEL
LIN {X 0,Y 183.793,Z 451.442,A -85,B 0,C 180,E1 -22405.614,E2 -22405.614} C_VEL
LIN {X 0,Y 183.864,Z 453.488,A -85,B 0,C 180,E1 -22408.098,E2 -22408.098} C_VEL
LIN {X 0,Y 184.186,Z 454.745,A -85,B 0,C 180,E1 -22410,E2 -22410} C_VEL
LIN {X 0,Y 183.591,Z 456.066,A -85,B 0,C 180,E1 -22414.069,E2 -22414.069} C_VEL
LIN {X 0,Y 182.891,Z 456.298,A -85,B 0,C 180,E1 -22415.899,E2 -22415.899} C_VEL
LIN {X 0,Y 181.296,Z 456.195,A -85,B 0,C 180,E1 -22417.703,E2 -22417.703} C_VEL
LIN {X 0,Y 177.904,Z 455.128,A -85,B 0,C 180,E1 -22421.354,E2 -22421.354} C_VEL
LIN {X 0,Y 177.34,Z 454.226,A -85,B 0,C 180,E1 -22423.242,E2 -22423.242} C_VEL
LIN {X 0,Y 177.481,Z 453.879,A -85,B 0,C 180,E1 -22423.87,E2 -22423.87} C_VEL
LIN {X 0,Y 179.755,Z 450.95,A -85,B 0,C 180,E1 -22428.227,E2 -22428.227} C_VEL
LIN {X 0,Y 183.185,Z 446.366,A -85,B 0,C 180,E1 -22432.561,E2 -22432.561} C_VEL
LIN {X 0,Y 186.345,Z 441.805,A -85,B 0,C 180,E1 -22435.704,E2 -22435.704} C_VEL
LIN {X 0,Y 191.026,Z 435.18,A -85,B 0,C 180,E1 -22439.175,E2 -22439.175} C_VEL
LIN {X 0,Y 195.728,Z 428.108,A -85,B 0,C 180,E1 -22441.981,E2 -22441.981} C_VEL
LIN {X 0,Y 198.399,Z 422.669,A -85,B 0,C 180,E1 -22443.913,E2 -22443.913} C_VEL
LIN {X 0,Y 201.348,Z 414.624,A -85,B 0,C 180,E1 -22446.6,E2 -22446.6} C_VEL
LIN {X 0,Y 203.616,Z 405.341,A -85,B 0,C 180,E1 -22449.527,E2 -22449.527} C_VEL
LIN {X 0,Y 204.983,Z 395.404,A -85,B 0,C 180,E1 -22452.648,E2 -22452.648} C_VEL
LIN {X 0,Y 205.347,Z 389.305,A -85,B 0,C 180,E1 -22454.617,E2 -22454.617} C_VEL
LIN {X 0,Y 204.568,Z 384.787,A -85,B 0,C 180,E1 -22456.598,E2 -22456.598} C_VEL
LIN {X 0,Y 202.731,Z 378.299,A -85,B 0,C 180,E1 -22460.107,E2 -22460.107} C_VEL
LIN {X 0,Y 201.187,Z 372.936,A -85,B 0,C 180,E1 -22463.569,E2 -22463.569} C_VEL
LIN {X 0,Y 199.182,Z 366.093,A -85,B 0,C 180,E1 -22470.397,E2 -22470.397} C_VEL
LIN {X 0,Y 198.803,Z 364.194,A -85,B 0,C 180,E1 -22474.898,E2 -22474.898} C_VEL
LIN {X 0,Y 199.116,Z 363.698,A -85,B 0,C 180,E1 -22477.154,E2 -22477.154} C_VEL
LIN {X 0,Y 200.644,Z 365.929,A -85,B 0,C 180,E1 -22483.726,E2 -22483.726} C_VEL
LIN {X 0,Y 201.701,Z 367.179,A -85,B 0,C 180,E1 -22485.883,E2 -22485.883} C_VEL
LIN {X 0,Y 203.96,Z 371.108,A -85,B 0,C 180,E1 -22490.079,E2 -22490.079} C_VEL
LIN {X 0,Y 206.343,Z 376.49,A -85,B 0,C 180,E1 -22494.135,E2 -22494.135} C_VEL
LIN {X 0,Y 207.442,Z 379.72,A -85,B 0,C 180,E1 -22496.114,E2 -22496.114} C_VEL
LIN {X 0,Y 208.653,Z 385.985,A -85,B 0,C 180,E1 -22499.375,E2 -22499.375} C_VEL
LIN {X 0,Y 208.984,Z 390.527,A -85,B 0,C 180,E1 -22501.445,E2 -22501.445} C_VEL
LIN {X 0,Y 208.696,Z 394.009,A -85,B 0,C 180,E1 -22502.895,E2 -22502.895} C_VEL
LIN {X 0,Y 203.857,Z 402.589,A -85,B 0,C 180,E1 -22505.324,E2 -22505.324} C_VEL
LIN {X 0,Y 198.752,Z 410.41,A -85,B 0,C 180,E1 -22508.131,E2 -22508.131} C_VEL
LIN {X 0,Y 193.596,Z 417.376,A -85,B 0,C 180,E1 -22511.428,E2 -22511.428} C_VEL
LIN {X 0,Y 188.912,Z 422.913,A -85,B 0,C 180,E1 -22515.095,E2 -22515.095} C_VEL
LIN {X 0,Y 185.33,Z 426.6,A -85,B 0,C 180,E1 -22518.55,E2 -22518.55} C_VEL
LIN {X 0,Y 181.935,Z 429.473,A -85,B 0,C 180,E1 -22522.724,E2 -22522.724} C_VEL
LIN {X 0,Y 179.877,Z 430.634,A -85,B 0,C 180,E1 -22526.02,E2 -22526.02} C_VEL
LIN {X 0,Y 178.151,Z 430.932,A -85,B 0,C 180,E1 -22529.785,E2 -22529.785} C_VEL
LIN {X 0,Y 177.027,Z 430.093,A -85,B 0,C 180,E1 -22533.766,E2 -22533.766} C_VEL
LIN {X 0,Y 176.514,Z 428.395,A -85,B 0,C 180,E1 -22537.22,E2 -22537.22} C_VEL
LIN {X 0,Y 176.496,Z 425.636,A -85,B 0,C 180,E1 -22540.837,E2 -22540.837} C_VEL
LIN {X 0,Y 176.939,Z 421.902,A -85,B 0,C 180,E1 -22544.36,E2 -22544.36} C_VEL
LIN {X 0,Y 177.742,Z 417.192,A -85,B 0,C 180,E1 -22547.763,E2 -22547.763} C_VEL
LIN {X 0,Y 179.049,Z 410.099,A -85,B 0,C 180,E1 -22551.724,E2 -22551.724} C_VEL
LIN {X 0,Y 180.827,Z 401.925,A -85,B 0,C 180,E1 -22555.293,E2 -22555.293} C_VEL
LIN {X 0,Y 182.689,Z 393.045,A -85,B 0,C 180,E1 -22558.369,E2 -22558.369} C_VEL
LIN {X 0,Y 184.785,Z 383.512,A -85,B 0,C 180,E1 -22561.017,E2 -22561.017} C_VEL
LIN {X 0,Y 186.953,Z 372.726,A -85,B 0,C 180,E1 -22563.431,E2 -22563.431} C_VEL
LIN {X 0,Y 188.046,Z 366.556,A -85,B 0,C 180,E1 -22564.583,E2 -22564.583} C_VEL
LIN {X 0,Y 186.63,Z 358.834,A -85,B 0,C 180,E1 -22566.121,E2 -22566.121} C_VEL
LIN {X 0,Y 183.685,Z 347.855,A -85,B 0,C 180,E1 -22568.096,E2 -22568.096} C_VEL
LIN {X 0,Y 179.414,Z 335.25,A -85,B 0,C 180,E1 -22570.073,E2 -22570.073} C_VEL
LIN {X 0,Y 178.535,Z 332.247,A -85,B 0,C 180,E1 -22570.547,E2 -22570.547} C_VEL
LIN {X 0,Y 178.589,Z 332.239,A -85,B 0,C 180,E1 -22574.01,E2 -22574.01} C_VEL
LIN {X 0,Y 178.834,Z 332.212,A -85,B 0,C 180,E1 -22579.257,E2 -22579.257} C_VEL
LIN {X 0,Y 178.904,Z 332.198,A -85,B 0,C 180,E1 -22583.232,E2 -22583.232} C_VEL
LIN {X 0,Y 179.151,Z 332.169,A -85,B 0,C 180,E1 -22587.752,E2 -22587.752} C_VEL
LIN {X 0,Y 179.371,Z 332.137,A -85,B 0,C 180,E1 -22590,E2 -22590} C_VEL
LIN {X 0,Y 178.863,Z 332.206,A -85,B 0,C 180,E1 -22594.507,E2 -22594.507} C_VEL
LIN {X 0,Y 178.907,Z 332.199,A -85,B 0,C 180,E1 -22599.041,E2 -22599.041} C_VEL
LIN {X 0,Y 178.659,Z 332.227,A -85,B 0,C 180,E1 -22603.652,E2 -22603.652} C_VEL
LIN {X 0,Y 178.624,Z 332.233,A -85,B 0,C 180,E1 -22609.217,E2 -22609.217} C_VEL
LIN {X 0,Y 178.535,Z 332.244,A -85,B 0,C 180,E1 -22615.125,E2 -22615.125} C_VEL
LIN {X 0,Y 178.524,Z 332.244,A -85,B 0,C 180,E1 -22619.994,E2 -22619.994} C_VEL
LIN {X 0,Y 178.497,Z 332.251,A -85,B 0,C 180,E1 -22624.225,E2 -22624.225} C_VEL
LIN {X 0,Y 178.419,Z 332.255,A -85,B 0,C 180,E1 -22629.069,E2 -22629.069} C_VEL
LIN {X 0,Y 178.404,Z 332.263,A -85,B 0,C 180,E1 -22632.044,E2 -22632.044} C_VEL
LIN {X 0,Y 178.4,Z 332.26,A -85,B 0,C 180,E1 -22635.163,E2 -22635.163} C_VEL
LIN {X 0,Y 178.405,Z 332.26,A -85,B 0,C 180,E1 -22638.459,E2 -22638.459} C_VEL
LIN {X 0,Y 178.425,Z 332.257,A -85,B 0,C 180,E1 -22643.784,E2 -22643.784} C_VEL
LIN {X 0,Y 178.489,Z 332.249,A -85,B 0,C 180,E1 -22646.547,E2 -22646.547} C_VEL
LIN {X 0,Y 178.524,Z 332.246,A -85,B 0,C 180,E1 -22650.007,E2 -22650.007} C_VEL
LIN {X 0,Y 178.522,Z 332.245,A -85,B 0,C 180,E1 -22654.886,E2 -22654.886} C_VEL
LIN {X 0,Y 178.622,Z 332.232,A -85,B 0,C 180,E1 -22660.787,E2 -22660.787} C_VEL
LIN {X 0,Y 178.651,Z 332.23,A -85,B 0,C 180,E1 -22666.348,E2 -22666.348} C_VEL
LIN {X 0,Y 178.913,Z 332.197,A -85,B 0,C 180,E1 -22670.96,E2 -22670.96} C_VEL
LIN {X 0,Y 179.153,Z 332.164,A -85,B 0,C 180,E1 -22677.752,E2 -22677.752} C_VEL
LIN {X 0,Y 179.37,Z 332.14,A -85,B 0,C 180,E1 -22680,E2 -22680} C_VEL
LIN {X 0,Y 178.855,Z 332.205,A -85,B 0,C 180,E1 -22684.508,E2 -22684.508} C_VEL
LIN {X 0,Y 178.911,Z 332.199,A -85,B 0,C 180,E1 -22689.041,E2 -22689.041} C_VEL
LIN {X 0,Y 178.654,Z 332.226,A -85,B 0,C 180,E1 -22693.653,E2 -22693.653} C_VEL
LIN {X 0,Y 178.623,Z 332.233,A -85,B 0,C 180,E1 -22699.213,E2 -22699.213} C_VEL
LIN {X 0,Y 178.518,Z 332.231,A -85,B 0,C 180,E1 -22705.111,E2 -22705.111} C_VEL
LIN {X 0,Y 178.462,Z 332.253,A -85,B 0,C 180,E1 -22710.794,E2 -22710.794} C_VEL
LIN {X 0,Y 178.486,Z 332.255,A -85,B 0,C 180,E1 -22714.219,E2 -22714.219} C_VEL
LIN {X 0,Y 178.57,Z 332.329,A -85,B 0,C 180,E1 -22717.653,E2 -22717.653} C_VEL
LIN {X 0,Y 179.24,Z 335.914,A -85,B 0,C 180,E1 -22721.841,E2 -22721.841} C_VEL
LIN {X 0,Y 180.016,Z 340.061,A -85,B 0,C 180,E1 -22726.434,E2 -22726.434} C_VEL
LIN {X 0,Y 180.661,Z 343.285,A -85,B 0,C 180,E1 -22729.887,E2 -22729.887} C_VEL
LIN {X 0,Y 180.865,Z 344.89,A -85,B 0,C 180,E1 -22731.557,E2 -22731.557} C_VEL
LIN {X 0,Y 180.298,Z 347.588,A -85,B 0,C 180,E1 -22734.218,E2 -22734.218} C_VEL
LIN {X 0,Y 179.451,Z 350.515,A -85,B 0,C 180,E1 -22736.961,E2 -22736.961} C_VEL
LIN {X 0,Y 181.008,Z 364.289,A -85,B 0,C 180,E1 -22738.314,E2 -22738.314} C_VEL
LIN {X 0,Y 182.121,Z 377.54,A -85,B 0,C 180,E1 -22740.064,E2 -22740.064} C_VEL
LIN {X 0,Y 182.781,Z 390.344,A -85,B 0,C 180,E1 -22742.174,E2 -22742.174} C_VEL
LIN {X 0,Y 183.079,Z 401.374,A -85,B 0,C 180,E1 -22744.414,E2 -22744.414} C_VEL
LIN {X 0,Y 183.125,Z 410.204,A -85,B 0,C 180,E1 -22746.536,E2 -22746.536} C_VEL
LIN {X 0,Y 181.299,Z 418.863,A -85,B 0,C 180,E1 -22748.934,E2 -22748.934} C_VEL
LIN {X 0,Y 179.531,Z 427.149,A -85,B 0,C 180,E1 -22751.749,E2 -22751.749} C_VEL
LIN {X 0,Y 178.073,Z 435.155,A -85,B 0,C 180,E1 -22755.135,E2 -22755.135} C_VEL
LIN {X 0,Y 177.118,Z 441.569,A -85,B 0,C 180,E1 -22758.557,E2 -22758.557} C_VEL
LIN {X 0,Y 176.739,Z 446.631,A -85,B 0,C 180,E1 -22762,E2 -22762} C_VEL
LIN {X 0,Y 176.734,Z 450.488,A -85,B 0,C 180,E1 -22765.438,E2 -22765.438} C_VEL
LIN {X 0,Y 177.127,Z 453.908,A -85,B 0,C 180,E1 -22770,E2 -22770} C_VEL
LIN {X 0,Y 176.518,Z 455.483,A -85,B 0,C 180,E1 -22774.567,E2 -22774.567} C_VEL
LIN {X 0,Y 176.473,Z 455.447,A -85,B 0,C 180,E1 -22779.166,E2 -22779.166} C_VEL
LIN {X 0,Y 177.481,Z 453.879,A -85,B 0,C 180,E1 -22783.87,E2 -22783.87} C_VEL
LIN {X 0,Y 177.646,Z 452.828,A -85,B 0,C 180,E1 -22785.741,E2 -22785.741} C_VEL
LIN {X 0,Y 176.576,Z 450.645,A -85,B 0,C 180,E1 -22788.851,E2 -22788.851} C_VEL
LIN {X 0,Y 175.944,Z 448.571,A -85,B 0,C 180,E1 -22791.334,E2 -22791.334} C_VEL
LIN {X 0,Y 176.423,Z 446.741,A -85,B 0,C 180,E1 -22793.155,E2 -22793.155} C_VEL
LIN {X 0,Y 176.869,Z 446.062,A -85,B 0,C 180,E1 -22793.738,E2 -22793.738} C_VEL
LIN {X 0,Y 181.251,Z 440.391,A -85,B 0,C 180,E1 -22797.73,E2 -22797.73} C_VEL
LIN {X 0,Y 186.482,Z 433.492,A -85,B 0,C 180,E1 -22801.212,E2 -22801.212} C_VEL
LIN {X 0,Y 190.552,Z 427.59,A -85,B 0,C 180,E1 -22803.59,E2 -22803.59} C_VEL
LIN {X 0,Y 194.164,Z 420.076,A -85,B 0,C 180,E1 -22806.395,E2 -22806.395} C_VEL
LIN {X 0,Y 196.528,Z 413.305,A -85,B 0,C 180,E1 -22808.741,E2 -22808.741} C_VEL
LIN {X 0,Y 198.492,Z 405.972,A -85,B 0,C 180,E1 -22811.206,E2 -22811.206} C_VEL
LIN {X 0,Y 200.006,Z 397.287,A -85,B 0,C 180,E1 -22814.128,E2 -22814.128} C_VEL
LIN {X 0,Y 200.426,Z 393.459,A -85,B 0,C 180,E1 -22815.468,E2 -22815.468} C_VEL
LIN {X 0,Y 199.662,Z 388.218,A -85,B 0,C 180,E1 -22818.026,E2 -22818.026} C_VEL
LIN {X 0,Y 198.364,Z 382.979,A -85,B 0,C 180,E1 -22821.212,E2 -22821.212} C_VEL
LIN {X 0,Y 197.562,Z 379.013,A -85,B 0,C 180,E1 -22823.861,E2 -22823.861} C_VEL
LIN {X 0,Y 196.081,Z 373.066,A -85,B 0,C 180,E1 -22829.881,E2 -22829.881} C_VEL
LIN {X 0,Y 195.85,Z 371.599,A -85,B 0,C 180,E1 -22832.192,E2 -22832.192} C_VEL
LIN {X 0,Y 195.983,Z 370.193,A -85,B 0,C 180,E1 -22836.767,E2 -22836.767} C_VEL
LIN {X 0,Y 196.133,Z 370.523,A -85,B 0,C 180,E1 -22839.002,E2 -22839.002} C_VEL
LIN {X 0,Y 197.411,Z 372.341,A -85,B 0,C 180,E1 -22843.994,E2 -22843.994} C_VEL
LIN {X 0,Y 198.129,Z 373.244,A -85,B 0,C 180,E1 -22845.623,E2 -22845.623} C_VEL
LIN {X 0,Y 199.995,Z 377.005,A -85,B 0,C 180,E1 -22849.88,E2 -22849.88} C_VEL
LIN {X 0,Y 201.926,Z 382.139,A -85,B 0,C 180,E1 -22854.006,E2 -22854.006} C_VEL
LIN {X 0,Y 202.696,Z 385.263,A -85,B 0,C 180,E1 -22856.023,E2 -22856.023} C_VEL
LIN {X 0,Y 203.418,Z 390.648,A -85,B 0,C 180,E1 -22859.01,E2 -22859.01} C_VEL
LIN {X 0,Y 203.293,Z 395.749,A -85,B 0,C 180,E1 -22861.485,E2 -22861.485} C_VEL
LIN {X 0,Y 202.9,Z 397.032,A -85,B 0,C 180,E1 -22861.985,E2 -22861.985} C_VEL
LIN {X 0,Y 197.429,Z 405.769,A -85,B 0,C 180,E1 -22864.627,E2 -22864.627} C_VEL
LIN {X 0,Y 192.945,Z 412.006,A -85,B 0,C 180,E1 -22867.03,E2 -22867.03} C_VEL
LIN {X 0,Y 187.761,Z 418.446,A -85,B 0,C 180,E1 -22870.241,E2 -22870.241} C_VEL
LIN {X 0,Y 183.747,Z 422.964,A -85,B 0,C 180,E1 -22873.267,E2 -22873.267} C_VEL
LIN {X 0,Y 179.444,Z 427.062,A -85,B 0,C 180,E1 -22877.082,E2 -22877.082} C_VEL
LIN {X 0,Y 175.913,Z 429.809,A -85,B 0,C 180,E1 -22881.073,E2 -22881.073} C_VEL
LIN {X 0,Y 173.989,Z 430.937,A -85,B 0,C 180,E1 -22883.824,E2 -22883.824} C_VEL
LIN {X 0,Y 172.388,Z 431.483,A -85,B 0,C 180,E1 -22886.644,E2 -22886.644} C_VEL
LIN {X 0,Y 170.87,Z 431.365,A -85,B 0,C 180,E1 -22890.26,E2 -22890.26} C_VEL
LIN {X 0,Y 169.839,Z 430.238,A -85,B 0,C 180,E1 -22894.145,E2 -22894.145} C_VEL
LIN {X 0,Y 169.365,Z 427.765,A -85,B 0,C 180,E1 -22898.494,E2 -22898.494} C_VEL
LIN {X 0,Y 169.657,Z 423.589,A -85,B 0,C 180,E1 -22903.116,E2 -22903.116} C_VEL
LIN {X 0,Y 170.288,Z 419.409,A -85,B 0,C 180,E1 -22906.514,E2 -22906.514} C_VEL
LIN {X 0,Y 171.438,Z 413.121,A -85,B 0,C 180,E1 -22910.481,E2 -22910.481} C_VEL
LIN {X 0,Y 172.838,Z 406.253,A -85,B 0,C 180,E1 -22913.91,E2 -22913.91} C_VEL
LIN {X 0,Y 174.645,Z 398.146,A -85,B 0,C 180,E1 -22917.163,E2 -22917.163} C_VEL
LIN {X 0,Y 176.92,Z 388.212,A -85,B 0,C 180,E1 -22920.331,E2 -22920.331} C_VEL
LIN {X 0,Y 179.06,Z 378.205,A -85,B 0,C 180,E1 -22922.895,E2 -22922.895} C_VEL
LIN {X 0,Y 181.097,Z 367.65,A -85,B 0,C 180,E1 -22925.071,E2 -22925.071} C_VEL
LIN {X 0,Y 179.94,Z 360.903,A -85,B 0,C 180,E1 -22926.47,E2 -22926.47} C_VEL
LIN {X 0,Y 176.783,Z 349.117,A -85,B 0,C 180,E1 -22928.73,E2 -22928.73} C_VEL
LIN {X 0,Y 172.686,Z 336.869,A -85,B 0,C 180,E1 -22930.787,E2 -22930.787} C_VEL
LIN {X 0,Y 171.543,Z 333.139,A -85,B 0,C 180,E1 -22931.332,E2 -22931.332} C_VEL
LIN {X 0,Y 171.559,Z 333.116,A -85,B 0,C 180,E1 -22935.771,E2 -22935.771} C_VEL
LIN {X 0,Y 171.845,Z 333.084,A -85,B 0,C 180,E1 -22940.585,E2 -22940.585} C_VEL
LIN {X 0,Y 171.81,Z 333.085,A -85,B 0,C 180,E1 -22945.307,E2 -22945.307} C_VEL
LIN {X 0,Y 172.333,Z 333.014,A -85,B 0,C 180,E1 -22950,E2 -22950} C_VEL
LIN {X 0,Y 171.811,Z 333.085,A -85,B 0,C 180,E1 -22954.693,E2 -22954.693} C_VEL
LIN {X 0,Y 171.845,Z 333.078,A -85,B 0,C 180,E1 -22959.415,E2 -22959.415} C_VEL
LIN {X 0,Y 171.577,Z 333.11,A -85,B 0,C 180,E1 -22964.227,E2 -22964.227} C_VEL
LIN {X 0,Y 171.545,Z 333.115,A -85,B 0,C 180,E1 -22969.562,E2 -22969.562} C_VEL
LIN {X 0,Y 171.47,Z 333.125,A -85,B 0,C 180,E1 -22975.617,E2 -22975.617} C_VEL
LIN {X 0,Y 171.442,Z 333.125,A -85,B 0,C 180,E1 -22980.587,E2 -22980.587} C_VEL
LIN {X 0,Y 171.407,Z 333.132,A -85,B 0,C 180,E1 -22985.032,E2 -22985.032} C_VEL
LIN {X 0,Y 171.381,Z 333.131,A -85,B 0,C 180,E1 -22988.817,E2 -22988.817} C_VEL
LIN {X 0,Y 171.328,Z 333.142,A -85,B 0,C 180,E1 -22994.215,E2 -22994.215} C_VEL
LIN {X 0,Y 171.337,Z 333.14,A -85,B 0,C 180,E1 -22998.982,E2 -22998.982} C_VEL
LIN {X 0,Y 171.386,Z 333.135,A -85,B 0,C 180,E1 -23002.041,E2 -23002.041} C_VEL
LIN {X 0,Y 171.401,Z 333.13,A -85,B 0,C 180,E1 -23005.092,E2 -23005.092} C_VEL
LIN {X 0,Y 171.451,Z 333.126,A -85,B 0,C 180,E1 -23010.535,E2 -23010.535} C_VEL
LIN {X 0,Y 171.445,Z 333.129,A -85,B 0,C 180,E1 -23015.8,E2 -23015.8} C_VEL
LIN {X 0,Y 171.578,Z 333.109,A -85,B 0,C 180,E1 -23020.872,E2 -23020.872} C_VEL
LIN {X 0,Y 171.569,Z 333.113,A -85,B 0,C 180,E1 -23025.772,E2 -23025.772} C_VEL
LIN {X 0,Y 171.85,Z 333.075,A -85,B 0,C 180,E1 -23030.585,E2 -23030.585} C_VEL
LIN {X 0,Y 171.815,Z 333.081,A -85,B 0,C 180,E1 -23035.308,E2 -23035.308} C_VEL
LIN {X 0,Y 172.332,Z 333.016,A -85,B 0,C 180,E1 -23040,E2 -23040} C_VEL
LIN {X 0,Y 171.804,Z 333.082,A -85,B 0,C 180,E1 -23044.693,E2 -23044.693} C_VEL
LIN {X 0,Y 171.848,Z 333.078,A -85,B 0,C 180,E1 -23049.415,E2 -23049.415} C_VEL
LIN {X 0,Y 171.571,Z 333.109,A -85,B 0,C 180,E1 -23054.228,E2 -23054.228} C_VEL
LIN {X 0,Y 171.541,Z 333.115,A -85,B 0,C 180,E1 -23059.557,E2 -23059.557} C_VEL
LIN {X 0,Y 171.446,Z 333.111,A -85,B 0,C 180,E1 -23065.599,E2 -23065.599} C_VEL
LIN {X 0,Y 171.419,Z 333.129,A -85,B 0,C 180,E1 -23070.573,E2 -23070.573} C_VEL
LIN {X 0,Y 171.479,Z 333.124,A -85,B 0,C 180,E1 -23076.462,E2 -23076.462} C_VEL
LIN {X 0,Y 171.556,Z 333.306,A -85,B 0,C 180,E1 -23077.545,E2 -23077.545} C_VEL
LIN {X 0,Y 172.35,Z 337.655,A -85,B 0,C 180,E1 -23082.777,E2 -23082.777} C_VEL
LIN {X 0,Y 173.337,Z 342.443,A -85,B 0,C 180,E1 -23088.263,E2 -23088.263} C_VEL
LIN {X 0,Y 173.782,Z 345.408,A -85,B 0,C 180,E1 -23091.488,E2 -23091.488} C_VEL
LIN {X 0,Y 173.134,Z 348.117,A -85,B 0,C 180,E1 -23094.279,E2 -23094.279} C_VEL
LIN {X 0,Y 172.576,Z 349.877,A -85,B 0,C 180,E1 -23096.079,E2 -23096.079} C_VEL
LIN {X 0,Y 174.129,Z 363.871,A -85,B 0,C 180,E1 -23097.525,E2 -23097.525} C_VEL
LIN {X 0,Y 175.21,Z 377.563,A -85,B 0,C 180,E1 -23099.408,E2 -23099.408} C_VEL
LIN {X 0,Y 175.834,Z 390.08,A -85,B 0,C 180,E1 -23101.562,E2 -23101.562} C_VEL
LIN {X 0,Y 176.087,Z 401.365,A -85,B 0,C 180,E1 -23103.958,E2 -23103.958} C_VEL
LIN {X 0,Y 175.947,Z 411.203,A -85,B 0,C 180,E1 -23106.457,E2 -23106.457} C_VEL
LIN {X 0,Y 173.784,Z 420.593,A -85,B 0,C 180,E1 -23109.276,E2 -23109.276} C_VEL
LIN {X 0,Y 172.189,Z 428.381,A -85,B 0,C 180,E1 -23112.174,E2 -23112.174} C_VEL
LIN {X 0,Y 170.775,Z 435.994,A -85,B 0,C 180,E1 -23115.704,E2 -23115.704} C_VEL
LIN {X 0,Y 169.954,Z 442.086,A -85,B 0,C 180,E1 -23119.275,E2 -23119.275} C_VEL
LIN {X 0,Y 169.694,Z 446.891,A -85,B 0,C 180,E1 -23122.863,E2 -23122.863} C_VEL
LIN {X 0,Y 169.659,Z 450.496,A -85,B 0,C 180,E1 -23126.438,E2 -23126.438} C_VEL
LIN {X 0,Y 170.068,Z 453.054,A -85,B 0,C 180,E1 -23130,E2 -23130} C_VEL
LIN {X 0,Y 169.435,Z 454.777,A -85,B 0,C 180,E1 -23134.759,E2 -23134.759} C_VEL
LIN {X 0,Y 169.293,Z 455.051,A -85,B 0,C 180,E1 -23137.154,E2 -23137.154} C_VEL
LIN {X 0,Y 169.83,Z 454.429,A -85,B 0,C 180,E1 -23141.942,E2 -23141.942} C_VEL
LIN {X 0,Y 171.604,Z 452.365,A -85,B 0,C 180,E1 -23146.66,E2 -23146.66} C_VEL
LIN {X 0,Y 172.973,Z 450.785,A -85,B 0,C 180,E1 -23148.969,E2 -23148.969} C_VEL
LIN {X 0,Y 176.606,Z 446.404,A -85,B 0,C 180,E1 -23153.45,E2 -23153.45} C_VEL
LIN {X 0,Y 176.869,Z 446.062,A -85,B 0,C 180,E1 -23153.738,E2 -23153.738} C_VEL
LIN {X 0,Y 177.926,Z 443.977,A -85,B 0,C 180,E1 -23155.493,E2 -23155.493} C_VEL
LIN {X 0,Y 178.408,Z 440.303,A -85,B 0,C 180,E1 -23158.454,E2 -23158.454} C_VEL
LIN {X 0,Y 179.417,Z 436.08,A -85,B 0,C 180,E1 -23161.29,E2 -23161.29} C_VEL
LIN {X 0,Y 181.23,Z 433.143,A -85,B 0,C 180,E1 -23162.799,E2 -23162.799} C_VEL
LIN {X 0,Y 185.471,Z 427.175,A -85,B 0,C 180,E1 -23165.301,E2 -23165.301} C_VEL
LIN {X 0,Y 189.424,Z 419.103,A -85,B 0,C 180,E1 -23168.441,E2 -23168.441} C_VEL
LIN {X 0,Y 192.139,Z 411.671,A -85,B 0,C 180,E1 -23171.178,E2 -23171.178} C_VEL
LIN {X 0,Y 194.217,Z 403.711,A -85,B 0,C 180,E1 -23174.032,E2 -23174.032} C_VEL
LIN {X 0,Y 195.276,Z 398.308,A -85,B 0,C 180,E1 -23176.039,E2 -23176.039} C_VEL
LIN {X 0,Y 195.244,Z 395.134,A -85,B 0,C 180,E1 -23177.53,E2 -23177.53} C_VEL
LIN {X 0,Y 194.285,Z 389.047,A -85,B 0,C 180,E1 -23181.209,E2 -23181.209} C_VEL
LIN {X 0,Y 193.549,Z 384.533,A -85,B 0,C 180,E1 -23184.48,E2 -23184.48} C_VEL
LIN {X 0,Y 192.553,Z 379.974,A -85,B 0,C 180,E1 -23189.27,E2 -23189.27} C_VEL
LIN {X 0,Y 192.421,Z 378.234,A -85,B 0,C 180,E1 -23191.652,E2 -23191.652} C_VEL
LIN {X 0,Y 192.525,Z 376.553,A -85,B 0,C 180,E1 -23196.325,E2 -23196.325} C_VEL
LIN {X 0,Y 192.669,Z 376.632,A -85,B 0,C 180,E1 -23198.606,E2 -23198.606} C_VEL
LIN {X 0,Y 193.451,Z 378.055,A -85,B 0,C 180,E1 -23203.104,E2 -23203.104} C_VEL
LIN {X 0,Y 194.238,Z 379.121,A -85,B 0,C 180,E1 -23205.328,E2 -23205.328} C_VEL
LIN {X 0,Y 195.745,Z 382.672,A -85,B 0,C 180,E1 -23209.658,E2 -23209.658} C_VEL
LIN {X 0,Y 197.253,Z 387.57,A -85,B 0,C 180,E1 -23213.864,E2 -23213.864} C_VEL
LIN {X 0,Y 197.72,Z 390.607,A -85,B 0,C 180,E1 -23215.923,E2 -23215.923} C_VEL
LIN {X 0,Y 198.011,Z 395.78,A -85,B 0,C 180,E1 -23218.983,E2 -23218.983} C_VEL
LIN {X 0,Y 197.695,Z 398.763,A -85,B 0,C 180,E1 -23220.556,E2 -23220.556} C_VEL
LIN {X 0,Y 195.54,Z 402.329,A -85,B 0,C 180,E1 -23221.682,E2 -23221.682} C_VEL
LIN {X 0,Y 190.278,Z 409.753,A -85,B 0,C 180,E1 -23224.236,E2 -23224.236} C_VEL
LIN {X 0,Y 185.204,Z 416.045,A -85,B 0,C 180,E1 -23227.022,E2 -23227.022} C_VEL
LIN {X 0,Y 180.594,Z 421.123,A -85,B 0,C 180,E1 -23229.974,E2 -23229.974} C_VEL
LIN {X 0,Y 175.483,Z 426.003,A -85,B 0,C 180,E1 -23233.904,E2 -23233.904} C_VEL
LIN {X 0,Y 172.603,Z 428.406,A -85,B 0,C 180,E1 -23236.56,E2 -23236.56} C_VEL
LIN {X 0,Y 170.071,Z 430.172,A -85,B 0,C 180,E1 -23239.304,E2 -23239.304} C_VEL
LIN {X 0,Y 167.547,Z 431.551,A -85,B 0,C 180,E1 -23242.657,E2 -23242.657} C_VEL
LIN {X 0,Y 165.195,Z 432.153,A -85,B 0,C 180,E1 -23246.693,E2 -23246.693} C_VEL
LIN {X 0,Y 163.486,Z 431.611,A -85,B 0,C 180,E1 -23251.055,E2 -23251.055} C_VEL
LIN {X 0,Y 162.611,Z 430.206,A -85,B 0,C 180,E1 -23254.797,E2 -23254.797} C_VEL
LIN {X 0,Y 162.26,Z 427.734,A -85,B 0,C 180,E1 -23258.772,E2 -23258.772} C_VEL
LIN {X 0,Y 162.474,Z 424.282,A -85,B 0,C 180,E1 -23262.662,E2 -23262.662} C_VEL
LIN {X 0,Y 163.295,Z 419.044,A -85,B 0,C 180,E1 -23267.025,E2 -23267.025} C_VEL
LIN {X 0,Y 164.521,Z 412.55,A -85,B 0,C 180,E1 -23271.162,E2 -23271.162} C_VEL
LIN {X 0,Y 165.964,Z 405.814,A -85,B 0,C 180,E1 -23274.539,E2 -23274.539} C_VEL
LIN {X 0,Y 167.798,Z 397.743,A -85,B 0,C 180,E1 -23277.812,E2 -23277.812} C_VEL
LIN {X 0,Y 170.189,Z 387.65,A -85,B 0,C 180,E1 -23281.09,E2 -23281.09} C_VEL
LIN {X 0,Y 172.558,Z 376.725,A -85,B 0,C 180,E1 -23283.894,E2 -23283.894} C_VEL
LIN {X 0,Y 174.163,Z 368.773,A -85,B 0,C 180,E1 -23285.567,E2 -23285.567} C_VEL
LIN {X 0,Y 173.379,Z 363.548,A -85,B 0,C 180,E1 -23286.72,E2 -23286.72} C_VEL
LIN {X 0,Y 170.778,Z 353.31,A -85,B 0,C 180,E1 -23288.847,E2 -23288.847} C_VEL
LIN {X 0,Y 167.641,Z 343.224,A -85,B 0,C 180,E1 -23290.722,E2 -23290.722} C_VEL
LIN {X 0,Y 164.494,Z 333.995,A -85,B 0,C 180,E1 -23292.277,E2 -23292.277} C_VEL
LIN {X 0,Y 164.699,Z 333.971,A -85,B 0,C 180,E1 -23298.946,E2 -23298.946} C_VEL
LIN {X 0,Y 164.826,Z 333.956,A -85,B 0,C 180,E1 -23302.651,E2 -23302.651} C_VEL
LIN {X 0,Y 165.046,Z 333.926,A -85,B 0,C 180,E1 -23307.559,E2 -23307.559} C_VEL
LIN {X 0,Y 165.296,Z 333.89,A -85,B 0,C 180,E1 -23310,E2 -23310} C_VEL
LIN {X 0,Y 164.76,Z 333.963,A -85,B 0,C 180,E1 -23314.894,E2 -23314.894} C_VEL
LIN {X 0,Y 164.826,Z 333.95,A -85,B 0,C 180,E1 -23317.349,E2 -23317.349} C_VEL
LIN {X 0,Y 164.703,Z 333.969,A -85,B 0,C 180,E1 -23321.06,E2 -23321.06} C_VEL
LIN {X 0,Y 164.485,Z 333.995,A -85,B 0,C 180,E1 -23327.403,E2 -23327.403} C_VEL
LIN {X 0,Y 164.474,Z 333.997,A -85,B 0,C 180,E1 -23329.989,E2 -23329.989} C_VEL
LIN {X 0,Y 164.394,Z 334.008,A -85,B 0,C 180,E1 -23336.134,E2 -23336.134} C_VEL
LIN {X 0,Y 164.377,Z 334.005,A -85,B 0,C 180,E1 -23341.229,E2 -23341.229} C_VEL
LIN {X 0,Y 164.314,Z 334.014,A -85,B 0,C 180,E1 -23346.785,E2 -23346.785} C_VEL
LIN {X 0,Y 164.3,Z 334.016,A -85,B 0,C 180,E1 -23349.914,E2 -23349.914} C_VEL
LIN {X 0,Y 164.28,Z 334.021,A -85,B 0,C 180,E1 -23353.342,E2 -23353.342} C_VEL
LIN {X 0,Y 164.293,Z 334.013,A -85,B 0,C 180,E1 -23356.809,E2 -23356.809} C_VEL
LIN {X 0,Y 164.296,Z 334.019,A -85,B 0,C 180,E1 -23360.352,E2 -23360.352} C_VEL
LIN {X 0,Y 164.332,Z 334.01,A -85,B 0,C 180,E1 -23364.349,E2 -23364.349} C_VEL
LIN {X 0,Y 164.392,Z 334.008,A -85,B 0,C 180,E1 -23369.135,E2 -23369.135} C_VEL
LIN {X 0,Y 164.408,Z 334.002,A -85,B 0,C 180,E1 -23374.693,E2 -23374.693} C_VEL
LIN {X 0,Y 164.486,Z 333.992,A -85,B 0,C 180,E1 -23380.052,E2 -23380.052} C_VEL
LIN {X 0,Y 164.5,Z 333.995,A -85,B 0,C 180,E1 -23385.147,E2 -23385.147} C_VEL
LIN {X 0,Y 164.77,Z 333.956,A -85,B 0,C 180,E1 -23390.177,E2 -23390.177} C_VEL
LIN {X 0,Y 164.832,Z 333.952,A -85,B 0,C 180,E1 -23392.651,E2 -23392.651} C_VEL
LIN {X 0,Y 165.049,Z 333.921,A -85,B 0,C 180,E1 -23397.56,E2 -23397.56} C_VEL
LIN {X 0,Y 165.295,Z 333.893,A -85,B 0,C 180,E1 -23400,E2 -23400} C_VEL
LIN {X 0,Y 164.753,Z 333.958,A -85,B 0,C 180,E1 -23404.895,E2 -23404.895} C_VEL
LIN {X 0,Y 164.827,Z 333.951,A -85,B 0,C 180,E1 -23407.35,E2 -23407.35} C_VEL
LIN {X 0,Y 164.705,Z 333.967,A -85,B 0,C 180,E1 -23411.061,E2 -23411.061} C_VEL
LIN {X 0,Y 164.48,Z 333.995,A -85,B 0,C 180,E1 -23417.404,E2 -23417.404} C_VEL
LIN {X 0,Y 164.475,Z 333.996,A -85,B 0,C 180,E1 -23419.989,E2 -23419.989} C_VEL
LIN {X 0,Y 164.372,Z 333.988,A -85,B 0,C 180,E1 -23426.117,E2 -23426.117} C_VEL
LIN {X 0,Y 164.36,Z 334.009,A -85,B 0,C 180,E1 -23431.218,E2 -23431.218} C_VEL
LIN {X 0,Y 164.475,Z 334.018,A -85,B 0,C 180,E1 -23437.126,E2 -23437.126} C_VEL
LIN {X 0,Y 165.093,Z 337.304,A -85,B 0,C 180,E1 -23441.286,E2 -23441.286} C_VEL
LIN {X 0,Y 166.09,Z 342.372,A -85,B 0,C 180,E1 -23447.387,E2 -23447.387} C_VEL
LIN {X 0,Y 166.632,Z 345.31,A -85,B 0,C 180,E1 -23450.754,E2 -23450.754} C_VEL
LIN {X 0,Y 166.615,Z 346.675,A -85,B 0,C 180,E1 -23452.255,E2 -23452.255} C_VEL
LIN {X 0,Y 165.739,Z 349.379,A -85,B 0,C 180,E1 -23455.137,E2 -23455.137} C_VEL
LIN {X 0,Y 167.179,Z 362.692,A -85,B 0,C 180,E1 -23456.573,E2 -23456.573} C_VEL
LIN {X 0,Y 168.251,Z 375.911,A -85,B 0,C 180,E1 -23458.45,E2 -23458.45} C_VEL
LIN {X 0,Y 168.844,Z 388.695,A -85,B 0,C 180,E1 -23460.714,E2 -23460.714} C_VEL
LIN {X 0,Y 169.037,Z 399.782,A -85,B 0,C 180,E1 -23463.118,E2 -23463.118} C_VEL
LIN {X 0,Y 169.011,Z 410.607,A -85,B 0,C 180,E1 -23465.971,E2 -23465.971} C_VEL
LIN {X 0,Y 166.741,Z 420.3,A -85,B 0,C 180,E1 -23469.006,E2 -23469.006} C_VEL
LIN {X 0,Y 164.807,Z 429.395,A -85,B 0,C 180,E1 -23472.632,E2 -23472.632} C_VEL
LIN {X 0,Y 163.48,Z 436.702,A -85,B 0,C 180,E1 -23476.323,E2 -23476.323} C_VEL
LIN {X 0,Y 162.798,Z 442.556,A -85,B 0,C 180,E1 -23480.056,E2 -23480.056} C_VEL
LIN {X 0,Y 162.609,Z 447.079,A -85,B 0,C 180,E1 -23483.758,E2 -23483.758} C_VEL
LIN {X 0,Y 162.64,Z 450.502,A -85,B 0,C 180,E1 -23487.523,E2 -23487.523} C_VEL
LIN {X 0,Y 163.009,Z 452.2,A -85,B 0,C 180,E1 -23490,E2 -23490} C_VEL
LIN {X 0,Y 162.343,Z 454.041,A -85,B 0,C 180,E1 -23494.967,E2 -23494.967} C_VEL
LIN {X 0,Y 162.415,Z 454.373,A -85,B 0,C 180,E1 -23499.968,E2 -23499.968} C_VEL
LIN {X 0,Y 163.592,Z 453.201,A -85,B 0,C 180,E1 -23504.938,E2 -23504.938} C_VEL
LIN {X 0,Y 166.234,Z 450.585,A -85,B 0,C 180,E1 -23509.769,E2 -23509.769} C_VEL
LIN {X 0,Y 170.079,Z 446.469,A -85,B 0,C 180,E1 -23514.408,E2 -23514.408} C_VEL
LIN {X 0,Y 174.999,Z 440.642,A -85,B 0,C 180,E1 -23518.811,E2 -23518.811} C_VEL
LIN {X 0,Y 180.476,Z 434.092,A -85,B 0,C 180,E1 -23522.374,E2 -23522.374} C_VEL
LIN {X 0,Y 181.23,Z 433.143,A -85,B 0,C 180,E1 -23522.799,E2 -23522.799} C_VEL
LIN {X 0,Y 183.013,Z 430.098,A -85,B 0,C 180,E1 -23524.283,E2 -23524.283} C_VEL
LIN {X 0,Y 183.77,Z 427.179,A -85,B 0,C 180,E1 -23525.884,E2 -23525.884} C_VEL
LIN {X 0,Y 184.66,Z 419.137,A -85,B 0,C 180,E1 -23530.228,E2 -23530.228} C_VEL
LIN {X 0,Y 185.429,Z 416.807,A -85,B 0,C 180,E1 -23531.22,E2 -23531.22} C_VEL
LIN {X 0,Y 188.154,Z 409.406,A -85,B 0,C 180,E1 -23534.088,E2 -23534.088} C_VEL
LIN {X 0,Y 190.123,Z 402.18,A -85,B 0,C 180,E1 -23536.927,E2 -23536.927} C_VEL
LIN {X 0,Y 190.241,Z 399.453,A -85,B 0,C 180,E1 -23538.32,E2 -23538.32} C_VEL
LIN {X 0,Y 189.656,Z 393.852,A -85,B 0,C 180,E1 -23541.997,E2 -23541.997} C_VEL
LIN {X 0,Y 189.328,Z 390.272,A -85,B 0,C 180,E1 -23544.752,E2 -23544.752} C_VEL
LIN {X 0,Y 188.599,Z 384.755,A -85,B 0,C 180,E1 -23551.024,E2 -23551.024} C_VEL
LIN {X 0,Y 188.616,Z 383.518,A -85,B 0,C 180,E1 -23553.44,E2 -23553.44} C_VEL
LIN {X 0,Y 188.724,Z 382.741,A -85,B 0,C 180,E1 -23555.818,E2 -23555.818} C_VEL
LIN {X 0,Y 188.908,Z 382.641,A -85,B 0,C 180,E1 -23558.449,E2 -23558.449} C_VEL
LIN {X 0,Y 189.831,Z 384.483,A -85,B 0,C 180,E1 -23564.279,E2 -23564.279} C_VEL
LIN {X 0,Y 190.594,Z 386.349,A -85,B 0,C 180,E1 -23567.218,E2 -23567.218} C_VEL
LIN {X 0,Y 191.528,Z 389.192,A -85,B 0,C 180,E1 -23570.495,E2 -23570.495} C_VEL
LIN {X 0,Y 192.336,Z 392.775,A -85,B 0,C 180,E1 -23573.706,E2 -23573.706} C_VEL
LIN {X 0,Y 192.527,Z 397.317,A -85,B 0,C 180,E1 -23576.861,E2 -23576.861} C_VEL
LIN {X 0,Y 192.155,Z 401.599,A -85,B 0,C 180,E1 -23579.476,E2 -23579.476} C_VEL
LIN {X 0,Y 186.454,Z 409.44,A -85,B 0,C 180,E1 -23582.16,E2 -23582.16} C_VEL
LIN {X 0,Y 180.862,Z 416.008,A -85,B 0,C 180,E1 -23585.016,E2 -23585.016} C_VEL
LIN {X 0,Y 175.654,Z 421.438,A -85,B 0,C 180,E1 -23588.114,E2 -23588.114} C_VEL
LIN {X 0,Y 170.419,Z 426.209,A -85,B 0,C 180,E1 -23591.899,E2 -23591.899} C_VEL
LIN {X 0,Y 167.12,Z 428.741,A -85,B 0,C 180,E1 -23594.706,E2 -23594.706} C_VEL
LIN {X 0,Y 163.247,Z 431.193,A -85,B 0,C 180,E1 -23598.713,E2 -23598.713} C_VEL
LIN {X 0,Y 159.907,Z 432.58,A -85,B 0,C 180,E1 -23603.3,E2 -23603.3} C_VEL
LIN {X 0,Y 157.859,Z 432.727,A -85,B 0,C 180,E1 -23607.074,E2 -23607.074} C_VEL
LIN {X 0,Y 156.283,Z 431.892,A -85,B 0,C 180,E1 -23611.303,E2 -23611.303} C_VEL
LIN {X 0,Y 155.328,Z 429.741,A -85,B 0,C 180,E1 -23616.029,E2 -23616.029} C_VEL
LIN {X 0,Y 155.234,Z 425.969,A -85,B 0,C 180,E1 -23621.092,E2 -23621.092} C_VEL
LIN {X 0,Y 155.722,Z 422.12,A -85,B 0,C 180,E1 -23624.816,E2 -23624.816} C_VEL
LIN {X 0,Y 156.565,Z 417.285,A -85,B 0,C 180,E1 -23628.506,E2 -23628.506} C_VEL
LIN {X 0,Y 157.743,Z 411.365,A -85,B 0,C 180,E1 -23632.137,E2 -23632.137} C_VEL
LIN {X 0,Y 159.647,Z 403.179,A -85,B 0,C 180,E1 -23636.147,E2 -23636.147} C_VEL
LIN {X 0,Y 161.853,Z 393.62,A -85,B 0,C 180,E1 -23639.818,E2 -23639.818} C_VEL
LIN {X 0,Y 164.165,Z 384.083,A -85,B 0,C 180,E1 -23642.74,E2 -23642.74} C_VEL
LIN {X 0,Y 166.498,Z 373.415,A -85,B 0,C 180,E1 -23645.365,E2 -23645.365} C_VEL
LIN {X 0,Y 167.281,Z 369.663,A -85,B 0,C 180,E1 -23646.148,E2 -23646.148} C_VEL
LIN {X 0,Y 166.424,Z 364.602,A -85,B 0,C 180,E1 -23647.335,E2 -23647.335} C_VEL
LIN {X 0,Y 163.411,Z 352.783,A -85,B 0,C 180,E1 -23649.875,E2 -23649.875} C_VEL
LIN {X 0,Y 159.186,Z 339.925,A -85,B 0,C 180,E1 -23652.33,E2 -23652.33} C_VEL
LIN {X 0,Y 157.42,Z 334.876,A -85,B 0,C 180,E1 -23653.214,E2 -23653.214} C_VEL
LIN {X 0,Y 157.687,Z 334.847,A -85,B 0,C 180,E1 -23659.73,E2 -23659.73} C_VEL
LIN {X 0,Y 157.763,Z 334.838,A -85,B 0,C 180,E1 -23662.32,E2 -23662.32} C_VEL
LIN {X 0,Y 158.258,Z 334.766,A -85,B 0,C 180,E1 -23670,E2 -23670} C_VEL
LIN {X 0,Y 157.764,Z 334.83,A -85,B 0,C 180,E1 -23677.68,E2 -23677.68} C_VEL
LIN {X 0,Y 157.637,Z 334.848,A -85,B 0,C 180,E1 -23681.237,E2 -23681.237} C_VEL
LIN {X 0,Y 157.454,Z 334.868,A -85,B 0,C 180,E1 -23685.534,E2 -23685.534} C_VEL
LIN {X 0,Y 157.371,Z 334.878,A -85,B 0,C 180,E1 -23690.933,E2 -23690.933} C_VEL
LIN {X 0,Y 157.316,Z 334.889,A -85,B 0,C 180,E1 -23696.685,E2 -23696.685} C_VEL
LIN {X 0,Y 157.279,Z 334.893,A -85,B 0,C 180,E1 -23702.427,E2 -23702.427} C_VEL
LIN {X 0,Y 157.284,Z 334.891,A -85,B 0,C 180,E1 -23706.457,E2 -23706.457} C_VEL
LIN {X 0,Y 157.213,Z 334.902,A -85,B 0,C 180,E1 -23712.11,E2 -23712.11} C_VEL
LIN {X 0,Y 157.211,Z 334.899,A -85,B 0,C 180,E1 -23717.89,E2 -23717.89} C_VEL
LIN {X 0,Y 157.269,Z 334.892,A -85,B 0,C 180,E1 -23723.551,E2 -23723.551} C_VEL
LIN {X 0,Y 157.295,Z 334.891,A -85,B 0,C 180,E1 -23728.096,E2 -23728.096} C_VEL
LIN {X 0,Y 157.317,Z 334.885,A -85,B 0,C 180,E1 -23733.465,E2 -23733.465} C_VEL
LIN {X 0,Y 157.393,Z 334.876,A -85,B 0,C 180,E1 -23739.67,E2 -23739.67} C_VEL
LIN {X 0,Y 157.437,Z 334.873,A -85,B 0,C 180,E1 -23744.465,E2 -23744.465} C_VEL
LIN {X 0,Y 157.691,Z 334.838,A -85,B 0,C 180,E1 -23749.731,E2 -23749.731} C_VEL
LIN {X 0,Y 157.769,Z 334.831,A -85,B 0,C 180,E1 -23752.32,E2 -23752.32} C_VEL
LIN {X 0,Y 158.257,Z 334.77,A -85,B 0,C 180,E1 -23760,E2 -23760} C_VEL
LIN {X 0,Y 157.765,Z 334.831,A -85,B 0,C 180,E1 -23767.68,E2 -23767.68} C_VEL
LIN {X 0,Y 157.639,Z 334.847,A -85,B 0,C 180,E1 -23771.236,E2 -23771.236} C_VEL
LIN {X 0,Y 157.439,Z 334.871,A -85,B 0,C 180,E1 -23775.536,E2 -23775.536} C_VEL
LIN {X 0,Y 157.368,Z 334.878,A -85,B 0,C 180,E1 -23780.933,E2 -23780.933} C_VEL
LIN {X 0,Y 157.311,Z 334.866,A -85,B 0,C 180,E1 -23786.681,E2 -23786.681} C_VEL
LIN {X 0,Y 157.278,Z 334.896,A -85,B 0,C 180,E1 -23792.427,E2 -23792.427} C_VEL
LIN {X 0,Y 157.444,Z 334.953,A -85,B 0,C 180,E1 -23797.012,E2 -23797.012} C_VEL
LIN {X 0,Y 158.122,Z 338.599,A -85,B 0,C 180,E1 -23801.813,E2 -23801.813} C_VEL
LIN {X 0,Y 158.904,Z 342.59,A -85,B 0,C 180,E1 -23806.82,E2 -23806.82} C_VEL
LIN {X 0,Y 159.497,Z 345.52,A -85,B 0,C 180,E1 -23810.33,E2 -23810.33} C_VEL
LIN {X 0,Y 159.395,Z 347.432,A -85,B 0,C 180,E1 -23812.529,E2 -23812.529} C_VEL
LIN {X 0,Y 158.896,Z 348.864,A -85,B 0,C 180,E1 -23814.134,E2 -23814.134} C_VEL
LIN {X 0,Y 160.356,Z 362.405,A -85,B 0,C 180,E1 -23815.676,E2 -23815.676} C_VEL
LIN {X 0,Y 161.391,Z 376.171,A -85,B 0,C 180,E1 -23817.727,E2 -23817.727} C_VEL
LIN {X 0,Y 161.88,Z 388.173,A -85,B 0,C 180,E1 -23819.965,E2 -23819.965} C_VEL
LIN {X 0,Y 162.032,Z 399.564,A -85,B 0,C 180,E1 -23822.558,E2 -23822.558} C_VEL
LIN {X 0,Y 162.021,Z 409.758,A -85,B 0,C 180,E1 -23825.365,E2 -23825.365} C_VEL
LIN {X 0,Y 160.569,Z 416.531,A -85,B 0,C 180,E1 -23827.481,E2 -23827.481} C_VEL
LIN {X 0,Y 158.326,Z 426.242,A -85,B 0,C 180,E1 -23831.227,E2 -23831.227} C_VEL
LIN {X 0,Y 156.808,Z 434.097,A -85,B 0,C 180,E1 -23835.066,E2 -23835.066} C_VEL
LIN {X 0,Y 155.969,Z 439.388,A -85,B 0,C 180,E1 -23838.301,E2 -23838.301} C_VEL
LIN {X 0,Y 155.595,Z 444.535,A -85,B 0,C 180,E1 -23842.212,E2 -23842.212} C_VEL
LIN {X 0,Y 155.556,Z 448.444,A -85,B 0,C 180,E1 -23846.114,E2 -23846.114} C_VEL
LIN {X 0,Y 155.95,Z 451.265,A -85,B 0,C 180,E1 -23850,E2 -23850} C_VEL
LIN {X 0,Y 155.442,Z 452.488,A -85,B 0,C 180,E1 -23852.591,E2 -23852.591} C_VEL
LIN {X 0,Y 155.255,Z 453.299,A -85,B 0,C 180,E1 -23855.194,E2 -23855.194} C_VEL
LIN {X 0,Y 155.389,Z 453.777,A -85,B 0,C 180,E1 -23860.423,E2 -23860.423} C_VEL
LIN {X 0,Y 156.702,Z 452.821,A -85,B 0,C 180,E1 -23865.611,E2 -23865.611} C_VEL
LIN {X 0,Y 159.535,Z 450.394,A -85,B 0,C 180,E1 -23870.636,E2 -23870.636} C_VEL
LIN {X 0,Y 163.611,Z 446.472,A -85,B 0,C 180,E1 -23875.44,E2 -23875.44} C_VEL
LIN {X 0,Y 167.407,Z 442.495,A -85,B 0,C 180,E1 -23878.868,E2 -23878.868} C_VEL
LIN {X 0,Y 171.974,Z 437.527,A -85,B 0,C 180,E1 -23882.091,E2 -23882.091} C_VEL
LIN {X 0,Y 178.129,Z 430.321,A -85,B 0,C 180,E1 -23885.589,E2 -23885.589} C_VEL
LIN {X 0,Y 181.873,Z 424.305,A -85,B 0,C 180,E1 -23888.191,E2 -23888.191} C_VEL
LIN {X 0,Y 185.109,Z 417.592,A -85,B 0,C 180,E1 -23890.913,E2 -23890.913} C_VEL
LIN {X 0,Y 185.429,Z 416.807,A -85,B 0,C 180,E1 -23891.22,E2 -23891.22} C_VEL
LIN {X 0,Y 186.364,Z 413.47,A -85,B 0,C 180,E1 -23892.703,E2 -23892.703} C_VEL
LIN {X 0,Y 186.49,Z 410.559,A -85,B 0,C 180,E1 -23894.302,E2 -23894.302} C_VEL
LIN {X 0,Y 185.581,Z 405.568,A -85,B 0,C 180,E1 -23897.696,E2 -23897.696} C_VEL
LIN {X 0,Y 185.083,Z 402.347,A -85,B 0,C 180,E1 -23900.006,E2 -23900.006} C_VEL
LIN {X 0,Y 184.859,Z 398.325,A -85,B 0,C 180,E1 -23902.977,E2 -23902.977} C_VEL
LIN {X 0,Y 184.823,Z 395.538,A -85,B 0,C 180,E1 -23905.223,E2 -23905.223} C_VEL
LIN {X 0,Y 184.483,Z 390.576,A -85,B 0,C 180,E1 -23911.188,E2 -23911.188} C_VEL
LIN {X 0,Y 184.71,Z 388.589,A -85,B 0,C 180,E1 -23915.948,E2 -23915.948} C_VEL
LIN {X 0,Y 184.793,Z 388.493,A -85,B 0,C 180,E1 -23917.646,E2 -23917.646} C_VEL
LIN {X 0,Y 185.17,Z 389.474,A -85,B 0,C 180,E1 -23922.324,E2 -23922.324} C_VEL
LIN {X 0,Y 185.643,Z 390.291,A -85,B 0,C 180,E1 -23924.633,E2 -23924.633} C_VEL
LIN {X 0,Y 186.534,Z 393.323,A -85,B 0,C 180,E1 -23929.141,E2 -23929.141} C_VEL
LIN {X 0,Y 187.004,Z 396.135,A -85,B 0,C 180,E1 -23932.056,E2 -23932.056} C_VEL
LIN {X 0,Y 187.198,Z 399.126,A -85,B 0,C 180,E1 -23934.614,E2 -23934.614} C_VEL
LIN {X 0,Y 186.727,Z 403.662,A -85,B 0,C 180,E1 -23937.843,E2 -23937.843} C_VEL
LIN {X 0,Y 186.577,Z 404.487,A -85,B 0,C 180,E1 -23938.381,E2 -23938.381} C_VEL
LIN {X 0,Y 180.501,Z 412.041,A -85,B 0,C 180,E1 -23941.114,E2 -23941.114} C_VEL
LIN {X 0,Y 175.03,Z 417.905,A -85,B 0,C 180,E1 -23943.842,E2 -23943.842} C_VEL
LIN {X 0,Y 169.372,Z 423.21,A -85,B 0,C 180,E1 -23947.151,E2 -23947.151} C_VEL
LIN {X 0,Y 164.457,Z 427.232,A -85,B 0,C 180,E1 -23950.61,E2 -23950.61} C_VEL
LIN {X 0,Y 158.953,Z 430.918,A -85,B 0,C 180,E1 -23955.384,E2 -23955.384} C_VEL
LIN {X 0,Y 155.885,Z 432.421,A -85,B 0,C 180,E1 -23958.776,E2 -23958.776} C_VEL
LIN {X 0,Y 152.794,Z 433.304,A -85,B 0,C 180,E1 -23963.082,E2 -23963.082} C_VEL
LIN {X 0,Y 150.37,Z 433.072,A -85,B 0,C 180,E1 -23967.864,E2 -23967.864} C_VEL
LIN {X 0,Y 148.993,Z 431.918,A -85,B 0,C 180,E1 -23971.889,E2 -23971.889} C_VEL
LIN {X 0,Y 148.221,Z 429.709,A -85,B 0,C 180,E1 -23976.286,E2 -23976.286} C_VEL
LIN {X 0,Y 148.186,Z 425.642,A -85,B 0,C 180,E1 -23981.604,E2 -23981.604} C_VEL
LIN {X 0,Y 148.829,Z 420.878,A -85,B 0,C 180,E1 -23986.065,E2 -23986.065} C_VEL
LIN {X 0,Y 150.083,Z 414.559,A -85,B 0,C 180,E1 -23990.59,E2 -23990.59} C_VEL
LIN {X 0,Y 151.495,Z 407.987,A -85,B 0,C 180,E1 -23994.325,E2 -23994.325} C_VEL
LIN {X 0,Y 153.559,Z 399.429,A -85,B 0,C 180,E1 -23998.217,E2 -23998.217} C_VEL
LIN {X 0,Y 156.017,Z 389.53,A -85,B 0,C 180,E1 -24001.773,E2 -24001.773} C_VEL
LIN {X 0,Y 158.457,Z 379.209,A -85,B 0,C 180,E1 -24004.729,E2 -24004.729} C_VEL
LIN {X 0,Y 160.406,Z 370.345,A -85,B 0,C 180,E1 -24006.776,E2 -24006.776} C_VEL
LIN {X 0,Y 158.276,Z 360.396,A -85,B 0,C 180,E1 -24009.192,E2 -24009.192} C_VEL
LIN {X 0,Y 155.223,Z 349.794,A -85,B 0,C 180,E1 -24011.522,E2 -24011.522} C_VEL
LIN {X 0,Y 151.186,Z 338.253,A -85,B 0,C 180,E1 -24013.804,E2 -24013.804} C_VEL
LIN {X 0,Y 150.388,Z 335.752,A -85,B 0,C 180,E1 -24014.238,E2 -24014.238} C_VEL
LIN {X 0,Y 150.606,Z 335.728,A -85,B 0,C 180,E1 -24019.242,E2 -24019.242} C_VEL
LIN {X 0,Y 150.701,Z 335.717,A -85,B 0,C 180,E1 -24021.957,E2 -24021.957} C_VEL
LIN {X 0,Y 151.218,Z 335.642,A -85,B 0,C 180,E1 -24030,E2 -24030} C_VEL
LIN {X 0,Y 150.702,Z 335.71,A -85,B 0,C 180,E1 -24038.042,E2 -24038.042} C_VEL
LIN {X 0,Y 150.577,Z 335.728,A -85,B 0,C 180,E1 -24041.437,E2 -24041.437} C_VEL
LIN {X 0,Y 150.362,Z 335.754,A -85,B 0,C 180,E1 -24046.287,E2 -24046.287} C_VEL
LIN {X 0,Y 150.352,Z 335.753,A -85,B 0,C 180,E1 -24050.793,E2 -24050.793} C_VEL
